	xManualAuto:=ManualAuto, 
	xManualExtend:= 展缸2排液电池阀3手动, 
	xAutoExtend:= 展缸2排液电池阀3自动, 
	xReset:=复位  , 
	xPosExtend:=   , 
	xPosRetract:= , 
	tTimeout:= , 
	yValve1=> 展缸2排液电池阀3, 
	bAlarm=> );	
//展缸2排液电池阀4
cylinder_36(
    xManualRetract := , 
    xAutoRetract := , 
    yValve2 => , 
    cylinder_type :=0 , 

	xManualAuto:=ManualAuto, 
	xManualExtend:= 展缸2排液电池阀4手动, 
	xAutoExtend:= 展缸2排液电池阀4自动, 
	xReset:=复位  , 
	xPosExtend:=   , 
	xPosRetract:= , 
	tTimeout:= , 
	yValve1=> 展缸2排液电池阀4, 
	bAlarm=> );	
//展缸2吹气电池阀1
cylinder_37(
    xManualRetract := , 
    xAutoRetract := , 
    yValve2 => , 
    cylinder_type := 0, 

	xManualAuto:=ManualAuto, 
	xManualExtend:= 展缸2吹气电池阀1手动, 
	xAutoExtend:= 展缸2吹气电池阀1自动, 
	xReset:=复位  , 
	xPosExtend:=   , 
	xPosRetract:= , 
	tTimeout:= , 
	yValve1=> 展缸2吹气电池阀1, 
	bAlarm=> );	
//展缸2吹气电池阀2
cylinder_38(
    xManualRetract := , 
    xAutoRetract := , 
    yValve2 => , 
    cylinder_type := 0, 

	xManualAuto:=ManualAuto, 
	xManualExtend:= 展缸2吹气电池阀2手动, 
	xAutoExtend:= 展缸2吹气电池阀2自动, 
	xReset:=复位  , 
	xPosExtend:=   , 
	xPosRetract:= , 
	tTimeout:= , 
	yValve1=> 展缸2吹气电池阀2, 
	bAlarm=> );	
//展缸1吹气电池阀3
cylinder_39(
    xManualRetract := , 
    xAutoRetract := , 
    yValve2 => , 
    cylinder_type := 0, 

	xManualAuto:=ManualAuto, 
	xManualExtend:= 展缸2吹气电池阀3手动, 
	xAutoExtend:= 展缸2吹气电池阀3自动, 
	xReset:=复位  , 
	xPosExtend:=   , 
	xPosRetract:= , 
	tTimeout:= , 
	yValve1=> 展缸2吹气电池阀3, 
	bAlarm=> );	
//展缸2吹气电池阀4
cylinder_40(
    xManualRetract := , 
    xAutoRetract := , 
    yValve2 => , 
    cylinder_type := 0, 

	xManualAuto:=ManualAuto, 
	xManualExtend:= 展缸2吹气电池阀4手动, 
	xAutoExtend:= 展缸2吹气电池阀4自动, 
	xReset:=复位  , 
	xPosExtend:=   , 
	xPosRetract:= , 
	tTimeout:= , 
	yValve1=> 展缸2吹气电池阀4, 
	bAlarm=> );	
//收集进液电池阀
cylinder_41(
    xManualRetract := , 
    xAutoRetract := , 
    yValve2 => , 
    cylinder_type := 0, 

	xManualAuto:=ManualAuto, 
	xManualExtend:= 收集进液手动, 
	xAutoExtend:= 收集进液自动, 
	xReset:=复位  , 
	xPosExtend:=   , 
	xPosRetract:= , 
	tTimeout:= , 
	yValve1=> 收集平台进液2通电池阀, 
	bAlarm=> );	
//收集排液电池阀
cylinder_42(
    xManualRetract := , 
    xAutoRetract := , 
    yValve2 => , 
    cylinder_type := 0, 

	xManualAuto:=ManualAuto  , 
	xManualExtend:= 收集排液手动, 
	xAutoExtend:= 收集排液自动, 
	xReset:=复位  , 
	xPosExtend:=   , 
	xPosRetract:= , 
	tTimeout:= , 
	yValve1=> 收集平台排液3通电池阀, 
	bAlarm=> );	
//收集正压排液电池阀
cylinder_43(
    xManualRetract := , 
    xAutoRetract := , 
    yValve2 => , 
    cylinder_type :=0 , 

	xManualAuto:=ManualAuto  , 
	xManualExtend:= 收集正压排液手动, 
	xAutoExtend:= 收集正压排液自动, 
	xReset:=复位  , 
	xPosExtend:=   , 
	xPosRetract:= , 
	tTimeout:= , 
	yValve1=> 收集平台正压排液阀, 
	bAlarm=> );	
//溶液收集瓶定位气缸
cylinder_44(
    xManualRetract := , 
    xAutoRetract := , 
    yValve2 => , 
    cylinder_type := 0, 

	xManualAuto:=ManualAuto  , 
	xManualExtend:= 溶液收集瓶定位手动, 
	xAutoExtend:= 溶液收集瓶定位自动, 
	xReset:=复位  , 
	xPosExtend:=   , 
	xPosRetract:= , 
	tTimeout:= , 
	yValve1=> 溶液收集瓶工位定位气缸, 
	bAlarm=> );	
//上样定位气缸
cylinder_45(
    xManualRetract := , 
    xAutoRetract := , 
    yValve2 => , 
    cylinder_type :=0 , 

	xManualAuto:=ManualAuto  , 
	xManualExtend:= 上样定位手动, 
	xAutoExtend:= 上样定位自动, 
	xReset:=复位  , 
	xPosExtend:=   , 
	xPosRetract:= , 
	tTimeout:= , 
	yValve1=> 上样定位气缸, 
	bAlarm=> );	
//上样点样三通电池阀
cylinder_46(
    xManualRetract := , 
    xAutoRetract := , 
    yValve2 => , 
    cylinder_type :=0 , 

	xManualAuto:=ManualAuto  , 
	xManualExtend:= 上样点样三通电池阀手动, 
	xAutoExtend:= 上样点样三通电池阀自动, 
	xReset:=复位  , 
	xPosExtend:=   , 
	xPosRetract:= , 
	tTimeout:= , 
	yValve1=> 上样点样三通电池阀, 
	bAlarm=> );	
//刮板拍照真空泵
cylinder_46(
    xManualRetract := , 
    xAutoRetract := , 
    yValve2 => , 
    cylinder_type := 0, 

	xManualAuto:=ManualAuto  , 
	xManualExtend:=刮板拍照真空手动 , 
	xAutoExtend:= 刮板拍照真空自动, 
	xReset:=复位  , 
	xPosExtend:=   , 
	xPosRetract:= , 
	tTimeout:= , 
	yValve1=> 刮板拍照真空阀, 
	bAlarm=> );	
//刮板拍照无刷电机
cylinder_47(
    xManualRetract := , 
    xAutoRetract := , 
    yValve2 => , 
    cylinder_type :=0 , 

	xManualAuto:=ManualAuto  , 
	xManualExtend:=刮板拍照无刷电机手动 , 
	xAutoExtend:=刮板拍照无刷电机自动 , 
	xReset:=复位  , 
	xPosExtend:=   , 
	xPosRetract:= , 
	tTimeout:= , 
	yValve1=> 刮板拍照无刷电机, 
	bAlarm=> );	
//刮板拍照定位气缸
cylinder_48(
    xManualRetract := , 
    xAutoRetract := , 
    yValve2 => , 
    cylinder_type :=0 , 

	xManualAuto:=ManualAuto  , 
	xManualExtend:= 刮板拍照定位气缸手动, 
	xAutoExtend:=刮板拍照定位气缸自动 , 
	xReset:=复位  , 
	xPosExtend:=   , 
	xPosRetract:= , 
	tTimeout:= , 
	yValve1=> 刮板拍照定位气缸, 
	bAlarm=> );	
//粉末收集器定位气缸
cylinder_49(
    xManualRetract := , 
    xAutoRetract := , 
    yValve2 => , 
    cylinder_type :=0 , 

	xManualAuto:=ManualAuto  , 
	xManualExtend:= 粉末收集器定位手动, 
	xAutoExtend:= 粉末收集器定位自动, 
	xReset:=复位  , 
	xPosExtend:=   , 
	xPosRetract:= , 
	tTimeout:= , 
	yValve1=> 粉末收集器工位定位气缸, 
	bAlarm=> );	
//上样吹气电池阀
cylinder_50(
    xManualRetract := , 
    xAutoRetract := , 
    yValve2 => , 
    cylinder_type := 0, 

	xManualAuto:=ManualAuto  , 
	xManualExtend:= 上样吹气手动, 
	xAutoExtend:= 上样吹气自动, 
	xReset:=复位  , 
	xPosExtend:=   , 
	xPosRetract:= , 
	tTimeout:= , 
	yValve1=> 上样吹气二通阀, 
	bAlarm=> );

END_PROGRAM

// Device/Application/25_FB_功能块/FB_cylinder
FUNCTION_BLOCK FB_cylinder
VAR_INPUT
    xManualAuto : BOOL := FALSE;  // 手自动模式：FALSE=手动，TRUE=自动
    xManualExtend : BOOL;  // 手动伸出
	// 手动缩回
	xManualRetract: BOOL;
    xAutoExtend : BOOL;  // 自动伸出
	// 自动缩回
	xAutoRetract: BOOL;
    xReset : BOOL;  // 复位按钮
    xPosExtend : BOOL;  // 伸出到位传感器
    xPosRetract : BOOL;  // 缩回到位传感器
    tTimeout : TIME := T#5S;  // 动作超时时间
END_VAR
VAR_OUTPUT
    yValve1 : BOOL;  // 电磁阀1输出：TRUE=伸出，FALSE=缩回
	// 电磁阀2输出：TRUE=伸出，FALSE=缩回
	yValve2: BOOL;
    bAlarm : BOOL;  // 报警输出
END_VAR
VAR
    bEnableCmd1 : BOOL;  // 有效的命令1
	// 有效的命令1
	bEnableCmd2: BOOL;
	tActionTimer: TON;// 动作定时器
END_VAR
VAR_INPUT
	// 气缸类型  0 单控  1双控
	cylinder_type: INT;
END_VAR



CASE cylinder_type OF
	0:     //单控电池阀
		//命令逻辑选择
		IF xManualAuto  THEN
			//自动模式，使用自动命令
			bEnableCmd1 :=xAutoExtend;
			ELSE
			//手动模式，使用手动命令
			bEnableCmd1 :=xManualExtend  ;
		END_IF
		//控制指令
		IF bEnableCmd1 THEN
			//开始伸出
			yValve1:=TRUE;
			ELSE
			//开始缩回
			yValve1 :=FALSE;
		END_IF
		
	
			tActionTimer(IN := (NOT xPosExtend AND NOT yValve1)  OR   (NOT xPosRetract AND yValve1), PT:=tTimeout );
			bAlarm :=tActionTimer .Q;
	
	1:        //双控电池阀
		//命令逻辑选择
		IF xManualAuto  THEN
			//自动模式，使用自动命令
			bEnableCmd1 :=xAutoExtend;
			bEnableCmd2 :=xAutoRetract;
		ELSE
			//手动模式，使用手动命令
			bEnableCmd1 :=xManualExtend;
			bEnableCmd2 :=xManualRetract;
		END_IF
		//伸出控制指令
		IF bEnableCmd1 THEN
			//开始伸出
			yValve1:=TRUE;
			yValve2:=FALSE;
		ELSE 
			yValve1:=FALSE;
		END_IF
		
		IF bEnableCmd2 THEN
			//开始缩回
			yValve2:=TRUE;
			yValve1:=FALSE;
		ELSE 
			yValve2:=FALSE;
		END_IF
		
			tActionTimer(IN := (NOT xPosExtend AND NOT yValve1)  OR   (NOT xPosRetract AND yValve2), PT:=tTimeout );
			bAlarm :=tActionTimer .Q;
		
END_CASE

IF xReset THEN
	bAlarm:=FALSE ;
END_IF

END_FUNCTION_BLOCK

// Device/Application/50_action/Rail_Sync
PROGRAM Rail_Sync
VAR
	i : INT;
END_VAR

(* 地轨 11Y 双源同步桥 (非动作派发器, 是 PC<->HMI 点位对账工具).
   原理: HMI_地轨轴11Y.position[] 是单 ExtensionObject struct, OPC 逐成员读写不可行
         -> 让 PLC 当桥, OPC 只暴露 flat 数组 (复用 *_ActPos 镜像同套路).
   每扫描无条件执行 (挂 PLC_MainPRG 无条件段, 与 ActPos 镜像同处; 勿放运行态 CASE).
   守恒: PUSH 纯 PLC 内存拷贝, 任一侧可触发; PULL 写真源恒为 PC, HMI 触发=请 PC 提交. *)

// (1) 常开镜像: HMI 教值 -> flat 只读镜像 (PC 经此读做 diff/pull, 不直访 struct)
FOR i := 1 TO 6 DO
	Rail_Pos_HMI[i] := HMI_地轨轴11Y.position[i];
END_FOR

// (2) 同步邮箱
CASE Rail_Sync_Req OF
	1:  (* PUSH: PC 真源 Rail_Pos_Target[] -> HMI 工作副本 position[] (PLC 写自己 struct, 无 OPC 限制) *)
		FOR i := 1 TO 6 DO
			HMI_地轨轴11Y.position[i] := Rail_Pos_Target[i];
		END_FOR
		Rail_Sync_Ack := 1;     (* 完成 *)
		Rail_Sync_Req := 0;     (* 清请求 *)

	2:  (* PULL: 收现场教值回真源. PLC 写不了 yaml, 更不可碰 Rail_Pos_Target (单写者=PC).
	          -> 仅亮邮箱待 PC 提交. PC 轮询见 Req=2 -> 读 Rail_Pos_HMI[] -> 限位校验/diff/确认
	             -> 写 points.yaml + 重算并写 Rail_Pos_Target[] -> 由 PC 置 Req:=0,Ack:=1 (失败 Ack:=3). *)
		Rail_Sync_Ack := 2;     (* 待 PC 提交 (PC 接手后由 PC 改写 Ack/Req) *)
END_CASE

END_PROGRAM

// Device/Application/50_action/PLC_Pump_泵管理
PROGRAM PLC_Pump_泵管理
VAR
END_VAR

(* 真空泵集中管理: 大真空泵线圈的唯一聚合点 (每扫描无条件调用).
   大真空泵站位[] 引用计数总线 -> 大真空泵自动 (经 FB_cylinder cylinder_8 驱动 大真空泵 %QX2.4).
   写者: [0..8]=Develop_TankDrain 排液自治; [11]=上位机 Pump_L2 显式真空; [9][10] 已退役. *)
大真空泵自动 := 大真空泵站位[0] OR 大真空泵站位[1] OR 大真空泵站位[2] OR 大真空泵站位[3]
	OR 大真空泵站位[4] OR 大真空泵站位[5] OR 大真空泵站位[6] OR 大真空泵站位[7]
	OR 大真空泵站位[8] OR 大真空泵站位[9] OR 大真空泵站位[10] OR 大真空泵站位[11];

END_PROGRAM

// Device/Application/40_Man/Develop_TankDrain
PROGRAM Develop_TankDrain
VAR
	// 循环索引
	i: INT;
	// 全局真空泵控制标志
	anyDraining: BOOL;
	// 全局真空泵控制标志
	展开step: INT;
	// 全局真空泵控制标志
	TON_3: TON;
	// 全局真空泵控制标志
	TON_4: TON;
	BlowTimer: ARRAY[1..8] OF TON;
	BlowDuration: TIME := TIME#30s0ms;
END_VAR




A50_Expand_liquid_discharge_排液();

ACTION A50_Expand_liquid_discharge_排液:

// ══════════════════════════════════════════════════════════════
// 排液控制程序（per-tank 并行 FSM，每扫描周期调用）
// ══════════════════════════════════════════════════════════════
// 程序名：PRG_TankDrain
// 文件名：plc_develop_drain.txt
// 职责：监控 Tank_Drain_Enable[1..8]，触发对应缸的 3 阶段排液流程
// 触发条件：Tank_Drain_Enable[i]=TRUE 且 Tank_State[i]=40
// 完成标志：Tank_Drain_Done[i]=TRUE, Tank_State[i]=99
// 复位方式：PC 写 Tank_Drain_Enable[i]=FALSE → 清 Done；
//           PC 写 Tank_State[i]=0 → 释放缸
// ══════════════════════════════════════════════════════════════
// 3 阶段排液时序（工程师已验证）：
//   Phase A — Draining(50)：开排液阀 + 真空泵，等待 DrainDuration
//   Phase B — BlowAir(55) ：追加开吹气阀，等待 BlowDuration
//   Phase C — CylinderRetract(60)：关所有阀 + 气缸退回，等待到位传感器
// ══════════════════════════════════════════════════════════════
// 硬件拓扑：
//   - 每缸有独立排液电磁阀、吹气电磁阀、气缸（伸出/退回）
//   - 真空泵（大真空泵）全局共享，anyDraining 引用计数式控制
//   - 排液气泡传感器按组共享（仅用于监控，不参与控制逻辑）
//   - 支持 8 缸完全并行排液（各缸 FSM 独立推进）
// ══════════════════════════════════════════════════════════════
// Tank_State 状态转换（排液相关）：
//   40 (Developing)      → 50 (Draining)        : Drain_Enable[i] 触发
//   50 (Draining)        → 55 (BlowAir)         : DrainTimer[i].Q
//   55 (BlowAir)         → 60 (CylinderRetract) : BlowTimer[i].Q
//   60 (CylinderRetract) → 99 (Done)            : 气缸到位传感器
//   99 (Done)            → 0  (Idle)            : PC 写 Tank_State=0
//   50/55/60             → 90 (Error)           : 急停
//   注：55/60 为 PLC 内部子状态，PC 只关心 Drain_Done（state 99）
// ══════════════════════════════════════════════════════════════
// 物理 IO 映射表（工程师变量名 → 缸索引）：
//   i=1: 展缸1排液电池阀1自动 / 展缸1吹气电池阀1自动 / 展缸1气缸1自动 / 展缸1气缸1动点
//   i=2: 展缸1排液电池阀2自动 / 展缸1吹气电池阀2自动 / 展缸1气缸2自动 / 展缸1气缸2动点
//   i=3: 展缸1排液电池阀3自动 / 展缸1吹气电池阀3自动 / 展缸1气缸3自动 / 展缸1气缸3动点
//   i=4: 展缸1排液电池阀4自动 / 展缸1吹气电池阀4自动 / 展缸1气缸4自动 / 展缸1气缸4动点
//   i=5: 展缸2排液电池阀1自动 / 展缸2吹气电池阀1自动 / 展缸2气缸1自动 / 展缸2气缸1动点
//   i=6: 展缸2排液电池阀2自动 / 展缸2吹气电池阀2自动 / 展缸2气缸2自动 / 展缸2气缸2动点
//   i=7: 展缸2排液电池阀3自动 / 展缸2吹气电池阀3自动 / 展缸2气缸3自动 / 展缸2气缸3动点
//   i=8: 展缸2排液电池阀4自动 / 展缸2吹气电池阀4自动 / 展缸2气缸4自动 / 展缸2气缸4动点
//   全局: 大真空泵自动
//   监控: 展缸1排液气泡传感器 / 展缸2排液气泡传感器
// ══════════════════════════════════════════════════════════════



// ══ 急停联锁：排液程序响应急停 ══
IF NOT 急停 THEN
    FOR i := 1 TO 8 DO
        // 急停时将所有排液中的缸（50/55/60）标记为 Error
        IF Tank_State[i] = 50 OR Tank_State[i] = 55 OR Tank_State[i] = 60 THEN
            Tank_State[i] := 90;
        END_IF
        // 停止所有定时器
        DrainTimer[i](IN := FALSE, PT := T#0S);
        BlowTimer[i](IN := FALSE, PT := T#0S);
        // 关闭所有排液阀和吹气阀
        CASE i OF
            1: 展缸1排液电池阀1自动 := FALSE; 展缸1吹气电池阀1自动 := FALSE;
            2: 展缸1排液电池阀2自动 := FALSE; 展缸1吹气电池阀2自动 := FALSE;
            3: 展缸1排液电池阀3自动 := FALSE; 展缸1吹气电池阀3自动 := FALSE;
            4: 展缸1排液电池阀4自动 := FALSE; 展缸1吹气电池阀4自动 := FALSE;
            5: 展缸2排液电池阀1自动 := FALSE; 展缸2吹气电池阀1自动 := FALSE;
            6: 展缸2排液电池阀2自动 := FALSE; 展缸2吹气电池阀2自动 := FALSE;
            7: 展缸2排液电池阀3自动 := FALSE; 展缸2吹气电池阀3自动 := FALSE;
            8: 展缸2排液电池阀4自动 := FALSE; 展缸2吹气电池阀4自动 := FALSE;
        END_CASE
    END_FOR
    // 关闭真空泵
    大真空泵站位[0] := FALSE;
    RETURN;
END_IF

// ══ 主循环：逐缸并行处理排液 FSM ══
FOR i := 1 TO 8 DO
 DrainTimer[i](IN := (Tank_State[i] = 50  AND  (i>4 AND 展缸2溶剂废液检测传感器)) OR (Tank_State[i] = 50 AND (i<5 AND 展缸1溶剂废液检测传感器)) , PT := DrainDuration);

 BlowTimer[i](IN := Tank_State[i] = 55, PT := BlowDuration);
 
    // ── 场景 1：PC 撤销 Drain_Enable → 复位 Done 标志（握手完成）──
    IF NOT Tank_Drain_Enable[i] THEN
        Tank_Drain_Done[i] := FALSE;
        DrainTimer[i](IN := FALSE, PT := T#0S);
        BlowTimer[i](IN := FALSE, PT := T#0S);
        // 注意：不主动修改 Tank_State，由 PC 写 0 释放
    // ── 场景 2：Drain_Enable=TRUE，缸处于 Developing(40)，启动排液 Phase A ──
    ELSIF Tank_Drain_Enable[i] AND Tank_State[i] = 40 THEN
        // 开启排液阀
		大真空泵站位[i] := TRUE;
        CASE i OF
            1: 展缸1排液电池阀1自动 := TRUE;
            2: 展缸1排液电池阀2自动 := TRUE;
            3: 展缸1排液电池阀3自动 := TRUE;
            4: 展缸1排液电池阀4自动 := TRUE;
            5: 展缸2排液电池阀1自动 := TRUE;
            6: 展缸2排液电池阀2自动 := TRUE;
            7: 展缸2排液电池阀3自动 := TRUE;
            8: 展缸2排液电池阀4自动 := TRUE;
        END_CASE
        // 推进状态至 Draining
        Tank_State[i] := 50;
    // ── 场景 3：Phase A — Draining(50)，排液阀开 + 真空泵运行，等待排液定时完成 ──
    ELSIF Tank_State[i] = 50 AND (i<5 AND 展缸1溶剂废液检测传感器) THEN
       
        IF DrainTimer[i].Q THEN
            // 排液定时完成，锁定并复位 DrainTimer
            DrainTimer[i](IN := FALSE, PT := T#0S);
            // 开启吹气阀（排液阀保持开启），进入 Phase B
            CASE i OF
                1: 展缸1吹气电池阀1自动 := TRUE;
                2: 展缸1吹气电池阀2自动 := TRUE;
                3: 展缸1吹气电池阀3自动 := TRUE;
                4: 展缸1吹气电池阀4自动 := TRUE;
                
            END_CASE
            Tank_State[i] := 55;
        END_IF
	ELSIF Tank_State[i] = 50  AND  (i>4AND 展缸2溶剂废液检测传感器) THEN
       
        IF DrainTimer[i].Q THEN
            // 排液定时完成，锁定并复位 DrainTimer
            DrainTimer[i](IN := FALSE, PT := T#0S);
            // 开启吹气阀（排液阀保持开启），进入 Phase B
            CASE i OF
                5: 展缸2吹气电池阀1自动 := TRUE;
                6: 展缸2吹气电池阀2自动 := TRUE;
                7: 展缸2吹气电池阀3自动 := TRUE;
                8: 展缸2吹气电池阀4自动 := TRUE;
            END_CASE
            Tank_State[i] := 55;
        END_IF
    // ── 场景 4：Phase B — BlowAir(55)，吹气阀开，等待吹气定时完成 ──
    ELSIF Tank_State[i] = 55 THEN
        大真空泵站位[i] := FALSE;
        IF BlowTimer[i].Q THEN
            // 吹气完成，锁定并复位 BlowTimer
            BlowTimer[i](IN := FALSE, PT := T#0S);
            // 关闭排液阀和吹气阀，启动气缸退回，进入 Phase C
            CASE i OF
                1: 展缸1排液电池阀1自动 := FALSE; 展缸1吹气电池阀1自动 := FALSE; 展缸1气缸1自动 := FALSE;
                2: 展缸1排液电池阀2自动 := FALSE; 展缸1吹气电池阀2自动 := FALSE; 展缸1气缸2自动 := FALSE;
                3: 展缸1排液电池阀3自动 := FALSE; 展缸1吹气电池阀3自动 := FALSE; 展缸1气缸3自动 := FALSE;
                4: 展缸1排液电池阀4自动 := FALSE; 展缸1吹气电池阀4自动 := FALSE; 展缸1气缸4自动 := FALSE;
                5: 展缸2排液电池阀1自动 := FALSE; 展缸2吹气电池阀1自动 := FALSE; 展缸2气缸1自动 := FALSE;
                6: 展缸2排液电池阀2自动 := FALSE; 展缸2吹气电池阀2自动 := FALSE; 展缸2气缸2自动 := FALSE;
                7: 展缸2排液电池阀3自动 := FALSE; 展缸2吹气电池阀3自动 := FALSE; 展缸2气缸3自动 := FALSE;
                8: 展缸2排液电池阀4自动 := FALSE; 展缸2吹气电池阀4自动 := FALSE; 展缸2气缸4自动 := FALSE;
            END_CASE
            Tank_State[i] := 60;
       END_IF
    // ── 场景 5：Phase C — CylinderRetract(60)，等待气缸退回到位 ──
    ELSIF Tank_State[i] = 60 THEN
        CASE i OF
            1: IF 展缸1气缸1原点 THEN   Tank_Drain_Done[1] := TRUE; Tank_State[1] := 99; END_IF
            2: IF 展缸1气缸2原点 THEN   Tank_Drain_Done[2] := TRUE; Tank_State[2] := 99; END_IF
            3: IF 展缸1气缸3原点 THEN   Tank_Drain_Done[3] := TRUE; Tank_State[3] := 99; END_IF
            4: IF 展缸1气缸4原点 THEN   Tank_Drain_Done[4] := TRUE; Tank_State[4] := 99; END_IF
            5: IF 展缸2气缸1原点 THEN   Tank_Drain_Done[5] := TRUE; Tank_State[5] := 99; END_IF
            6: IF 展缸2气缸2原点 THEN   Tank_Drain_Done[6] := TRUE; Tank_State[6] := 99; END_IF
            7: IF 展缸2气缸3原点 THEN   Tank_Drain_Done[7] := TRUE; Tank_State[7] := 99; END_IF
            8: IF 展缸2气缸4原点 THEN   Tank_Drain_Done[8] := TRUE; Tank_State[8] := 99; END_IF
        END_CASE
	END_IF
END_FOR
END_ACTION

END_PROGRAM

// Device/Application/50_action/Pump_L2
PROGRAM Pump_L2
VAR
	bActionDone: BOOL;
	bActionError: BOOL;
	L2_StartTrig: R_TRIG;
END_VAR

(* Pump 真空泵 L2 统一动作派发器 (独立真空泵原子动作通道).
   按 Pump_L2_ActionCode 派发: 10=真空泵开 / 20=真空泵关; 写上位机泵槽 大真空泵站位[11].
   实际线圈由 PLC_Pump_泵管理 聚合 大真空泵站位[] 驱动.
   Start 上升沿接受 -> RUNNING 调原子 -> bActionDone=DONE. *)
L2_StartTrig(CLK := Pump_L2_Start);

CASE Pump_L2_State OF
	0:  (* IDLE *)
		Pump_L2_Step := 0;
		IF L2_StartTrig.Q THEN
			Pump_L2_AcceptedSeq := Pump_L2_RequestSeq;
			Pump_L2_ActiveCode  := Pump_L2_ActionCode;
			Pump_L2_ErrorCode   := 0;
			Pump_L2_Retryable   := FALSE;
			bActionDone  := FALSE;
			bActionError := FALSE;
			CASE Pump_L2_ActionCode OF
				10, 20:
					Pump_L2_SafeState := 0;
					Pump_L2_State     := 10;   (* RUNNING *)
			ELSE
				Pump_L2_ErrorCode    := 101;  (* 未知动作码 *)
				Pump_L2_Retryable    := TRUE;
				Pump_L2_CompletedSeq := Pump_L2_AcceptedSeq;
				Pump_L2_State        := 30;   (* REJECTED *)
			END_CASE
		END_IF

	10: (* RUNNING *)
		IF Pump_L2_Reset THEN                (* RUNNING 中 RESET: 中止回 IDLE *)
			Pump_L2_State := 0;
		ELSE
			CASE Pump_L2_ActiveCode OF
				10: A10_vacuum_on();
				20: A20_vacuum_off();
			END_CASE
			IF bActionDone THEN
				bActionDone          := FALSE;
				Pump_L2_CompletedSeq := Pump_L2_AcceptedSeq;
				Pump_L2_State        := 20;   (* DONE *)
			ELSIF bActionError THEN
				bActionError         := FALSE;
				Pump_L2_Retryable    := TRUE;
				Pump_L2_CompletedSeq := Pump_L2_AcceptedSeq;
				Pump_L2_State        := 40;   (* ERROR *)
			END_IF
		END_IF

	20, 30, 40, 50:  (* 终态: 等 Start 落沿或 Reset 回 IDLE *)
		IF (NOT Pump_L2_Start) OR Pump_L2_Reset THEN
			Pump_L2_State := 0;
		END_IF
END_CASE

ACTION A10_vacuum_on:
(* 真空泵开: 置上位机泵槽 (实际线圈由 PLC_Pump_泵管理 聚合 大真空泵站位[] 驱动) *)
大真空泵站位[11] := TRUE;
bActionDone := TRUE;
END_ACTION

ACTION A20_vacuum_off:
(* 真空泵关: 清上位机泵槽 (排液 [0..8] 仍可独立保持真空) *)
大真空泵站位[11] := FALSE;
bActionDone := TRUE;
END_ACTION

END_PROGRAM

// Device/Application/50_action/Rail_L2
PROGRAM Rail_L2
VAR
	L2_StartTrig : R_TRIG;
	fTgt: LREAL;
END_VAR

(* 地轨 11Y L2 统一动作派发器 (第7通道).
   按位置码移地轨: Rail_L2_ActionCode=10 -> 移到 Rail_Pos_Target[Rail_Target_Position] (1..6, PC 真源).
   地轨坐标真源已收编为 PC 写的 Rail_Pos_Target[]; HMI position[] 降为手动示教工作副本, 自动不再读它.
   Start 上升沿接受 -> RUNNING 下发移动 -> bAbMoveDone=DONE. *)
L2_StartTrig(CLK := Rail_L2_Start);

CASE Rail_L2_State OF
	0:  (* IDLE *)
		Rail_L2_Step := 0;
		IF L2_StartTrig.Q THEN
			Rail_L2_AcceptedSeq := Rail_L2_RequestSeq;
			Rail_L2_ActiveCode  := Rail_L2_ActionCode;
			Rail_L2_ErrorCode   := 0;
			Rail_L2_Retryable   := FALSE;
// 			IF Rail_L2_ActionCode = 10
// 			   AND Rail_Target_Position >= 1 AND Rail_Target_Position <= 6 THEN
// 				Rail_L2_SafeState := 0;
// // 				地轨轴11YDATE.fAbsTarget := HMI_地轨轴11Y.position[Rail_Target_Position];
// 				地轨轴11YDATE.fAbsTarget := Rail_Pos_Target[Rail_Target_Position];
// 				地轨轴11YDATE.xMoveAbs   := TRUE;
// 				Rail_L2_State := 10;   (* RUNNING *)
// 			ELSE
// 				Rail_L2_ErrorCode    := 101;  (* 未知动作码 / 非法位置码 *)
// 				Rail_L2_Retryable    := TRUE;
// 				Rail_L2_CompletedSeq := Rail_L2_AcceptedSeq;
// 				Rail_L2_State        := 30;   (* REJECTED *)
// 			END_IF
			IF Rail_L2_ActionCode = 10 AND Rail_Target_Position >= 1 AND Rail_Target_Position <= 6 THEN
				fTgt := Rail_Pos_Target[Rail_Target_Position];     (* PC 真源坐标 *)
				IF fTgt <= 0.0 OR fTgt > 3000.0 THEN
					(* 兜底: PC 未 push / 重启后 Rail_Pos_Target 归 0 / 越限 → 拒绝, 绝不移到 0 端 *)
					Rail_L2_ErrorCode    := 102;   (* 目标未初始化或越限 *)
					Rail_L2_Retryable    := TRUE;
					Rail_L2_CompletedSeq := Rail_L2_AcceptedSeq;
					Rail_L2_State        := 30;    (* REJECTED *)
				ELSE
					Rail_L2_SafeState        := 0;
					地轨轴11YDATE.fAbsTarget := fTgt;
					地轨轴11YDATE.xMoveAbs   := TRUE;
					Rail_L2_State            := 10; (* RUNNING *)
				END_IF
			ELSE
				Rail_L2_ErrorCode    := 101;   (* 未知动作码 / 非法位置码 *)
				Rail_L2_Retryable    := TRUE;
				Rail_L2_CompletedSeq := Rail_L2_AcceptedSeq;
				Rail_L2_State        := 30;    (* REJECTED *)
END_IF
		END_IF

	10: (* RUNNING *)
		IF Rail_L2_Reset THEN                 (* RUNNING 中 RESET: 中止回 IDLE *)
			地轨轴11YDATE.xMoveAbs := FALSE;
			Rail_L2_State := 0;
		ELSIF 地轨轴11YDATE.bAbMoveDone THEN
			地轨轴11YDATE.xMoveAbs   := FALSE;
			Rail_L2_CompletedSeq := Rail_L2_AcceptedSeq;
			Rail_L2_State        := 20;   (* DONE *)
		END_IF
		(* 如地轨伺服有报警位, 在此 ELSIF <报警> THEN 置 Rail_L2_ErrorCode + State:=40 *)

	20, 30, 40, 50:  (* 终态: 等 Start 落沿或 Reset 回 IDLE *)
		IF (NOT Rail_L2_Start) OR Rail_L2_Reset THEN
			Rail_L2_State := 0;
		END_IF
END_CASE

END_PROGRAM

// Device/Application/50_action/FeedLift_L2
PROGRAM FeedLift_L2
VAR
	上料step: INT;
	下料step: INT;
	bActionDone: BOOL;
	bActionError: BOOL;
	L2_StartTrig: R_TRIG;
	feedlift_TO: TON;
END_VAR

(* FeedLift 工位 L2 统一动作派发器
   按 FeedLift_L2_ActionCode 派发到纯设备原子动作 (不含机器人/相机/CNC 握手).
   Start 上升沿接受请求 -> RUNNING 每周期调用对应原子 -> bActionDone=DONE / bActionError=ERROR. *)
L2_StartTrig(CLK := FeedLift_L2_Start);

CASE FeedLift_L2_State OF
	0:  (* IDLE *)
		FeedLift_L2_Step := 0;
		IF L2_StartTrig.Q THEN
			FeedLift_L2_AcceptedSeq := FeedLift_L2_RequestSeq;
			FeedLift_L2_ActiveCode  := FeedLift_L2_ActionCode;
			FeedLift_L2_ErrorCode   := 0;
			FeedLift_L2_Retryable   := FALSE;
			bActionDone  := FALSE;
			bActionError := FALSE;
			上料step := 0;
			下料step := 0;
			CASE FeedLift_L2_ActionCode OF
				11, 12, 21, 22:
					FeedLift_L2_SafeState := 0;
					FeedLift_L2_State     := 10;   (* RUNNING *)
			ELSE
				FeedLift_L2_ErrorCode    := 101;  (* 未知动作码 *)
				FeedLift_L2_Retryable    := TRUE;
				FeedLift_L2_CompletedSeq := FeedLift_L2_AcceptedSeq;
				FeedLift_L2_State        := 30;   (* REJECTED *)
			END_CASE
		END_IF

	10: (* RUNNING *)
		IF FeedLift_L2_Reset THEN FeedLift_L2_State := 0; RETURN; END_IF   (* RUNNING 中 RESET: 中止挂死动作 *)
		CASE FeedLift_L2_ActiveCode OF
			11: A11_feed_raise();
			12: A12_feed_lower();
			21: A21_unload_ready();
			22: A22_unload_bury();
		END_CASE
		IF bActionDone THEN
			bActionDone              := FALSE;
			FeedLift_L2_CompletedSeq := FeedLift_L2_AcceptedSeq;
			FeedLift_L2_State        := 20;   (* DONE *)
		ELSIF bActionError THEN              (* 设备预条件未满足 -> 报错交上位机 *)
			bActionError             := FALSE;
			FeedLift_L2_Retryable    := TRUE;
			FeedLift_L2_CompletedSeq := FeedLift_L2_AcceptedSeq;
			FeedLift_L2_State        := 40;   (* ERROR; ErrorCode 由原子置 *)
		END_IF

	20, 30, 40, 50:  (* 终态: 等 Start 落沿或 Reset 回 IDLE *)
		IF (NOT FeedLift_L2_Start) OR FeedLift_L2_Reset THEN
			FeedLift_L2_State := 0;
		END_IF
END_CASE

ACTION A11_feed_raise:
(* 上料: jog 上料Z1 升至取料光电 (上位机随后驱动机器人吸料); 无玻璃则报错交上位机 *)
feedlift_TO(IN:=上料step=0, PT:=T#10S);
CASE 上料step OF
	0:
		IF 玻璃上料轴1ZDATE.bHomed AND 玻璃升降接近开关1 AND 上料进料传感器 AND NOT Alarm.0 THEN
			上料step:=1;
		ELSIF feedlift_TO.Q THEN
			FeedLift_L2_ErrorCode:=301;   (* 上料无玻璃/传感器未就绪 *)
			上料step:=0;
			bActionError:=TRUE;
		END_IF
	1:
		IF 玻璃上料轴1ZDATE.fActPos>=510.0 AND 玻璃升降光电开关1 AND NOT 玻璃升降接近开关1 THEN
			Z1JOG_pos:=FALSE;
			Alarm.0:=TRUE;                       (* 上料机构无玻璃 *)
			上料step:=0;
			FeedLift_L2_ErrorCode:=301;
			bActionError:=TRUE;
		ELSIF NOT 玻璃升降光电开关1 AND 玻璃上料轴1ZDATE.fActPos<514 THEN
			Z1JOG_pos:=TRUE;
		ELSE
			Z1JOG_pos:=FALSE;
			上料step:=0;
			bActionDone:=TRUE;
		END_IF
END_CASE
END_ACTION

ACTION A22_unload_bury:
(* 下料: 机器人放废料后, jog Z2 下埋至光电消失 *)
feedlift_TO(IN:=下料step=0, PT:=T#10S);
CASE 下料step OF
	0:
		IF 玻璃升降光电开关2 AND 玻璃升降接近开关2 THEN
			Z2JOG_NEG:=TRUE;
			下料step:=10;
		ELSIF feedlift_TO.Q THEN
			FeedLift_L2_ErrorCode:=302;   (* 下料无玻璃/传感器未就绪 *)
			下料step:=0;
			bActionError:=TRUE;
		END_IF
	10:
		IF NOT 玻璃升降光电开关2 THEN
			Z2JOG_NEG:=FALSE;
			下料step:=0;
			bActionDone:=TRUE;
		END_IF
END_CASE
END_ACTION

ACTION A12_feed_lower:
(* 上料: 机器人吸住玻璃后, Z1 相对下降 5mm 让位 *)
CASE 上料step OF
	0:
		玻璃上料轴1ZDATE.fRelTarget:=-5.0;
		玻璃上料轴1ZDATE.xMoveRel:=TRUE;
		上料step:=10;
	10:
		IF 玻璃上料轴1ZDATE.bReMoveDone THEN
			玻璃上料轴1ZDATE.xMoveRel:=FALSE;
			上料step:=0;
			bActionDone:=TRUE;
		END_IF
END_CASE
END_ACTION

ACTION A21_unload_ready:
(* 下料: jog 下料Z2 到放废料位 (上位机随后驱动机器人放废料) *)
CASE 下料step OF
	0:
		IF 玻璃上料轴2ZDATE.bHomed AND 下料出料传感器 AND NOT Alarm.1 THEN
			下料step:=1;
		END_IF
	1:
		IF NOT 玻璃升降光电开关2 AND 玻璃上料轴2ZDATE.fActPos<510 THEN
			Z2JOG_POS:=TRUE;
		ELSE
			Z2JOG_POS:=FALSE;
			下料step:=10;
		END_IF
	10:
		IF 玻璃升降光电开关2 THEN
			Z2JOG_NEG:=TRUE;
			下料step:=15;
		END_IF
	15:
		IF NOT 玻璃升降光电开关2 THEN
			Z2JOG_NEG:=FALSE;
			下料step:=0;
			bActionDone:=TRUE;
		END_IF
END_CASE
END_ACTION

END_PROGRAM

// Device/Application/50_action/Sampling_L2
PROGRAM Sampling_L2
VAR
	初始化step: INT;
	清洗step: INT;
	清洗计数: INT;
	放硅胶板STEP: INT;
	上样准备step: INT;
	吸收液体step: INT;
	点样step: INT;
	喷涂移轴step: INT;
	N: INT;
	A: INT;
	打样伺服移动step: INT;
	spot_band_step: INT;
	spot_band_dry_count: INT;
	spot_band_old_6x_velocity: LREAL;
	spot_band_velocity_saved: BOOL;
	bActionDone: BOOL;
	bActionError: BOOL;
	TON_0: TON;
	TON_1: TON;
	L2_StartTrig: R_TRIG;
	R_TRIG: ARRAY[1..12] OF R_TRIG;
	TON: ARRAY[1..11] OF TON;
END_VAR

(* Sampling 工位 L2 统一动作派发器
   按 Sampling_L2_ActionCode 派发到纯设备原子动作 (不含机器人/相机/CNC 握手).
   Start 上升沿接受请求 -> RUNNING 每周期调用对应原子 -> bActionDone=DONE / bActionError=ERROR. *)
L2_StartTrig(CLK := Sampling_L2_Start);

CASE Sampling_L2_State OF
	0:  (* IDLE *)
		Sampling_L2_Step := 0;
		IF L2_StartTrig.Q THEN
			Sampling_L2_AcceptedSeq := Sampling_L2_RequestSeq;
			Sampling_L2_ActiveCode  := Sampling_L2_ActionCode;
			Sampling_L2_ErrorCode   := 0;
			Sampling_L2_Retryable   := FALSE;
			bActionDone  := FALSE;
			bActionError := FALSE;
			初始化step := 0;
			清洗step := 0;
			放硅胶板STEP := 0;
			上样准备step := 0;
			吸收液体step := 0;
			点样step := 0;
			喷涂移轴step := 0;
			spot_band_step := 0;
			spot_band_dry_count := 0;
			spot_band_velocity_saved := FALSE;
			CASE Sampling_L2_ActionCode OF
				10, 20, 31, 32, 33, 40, 50, 60, 61, 62:
					Sampling_L2_SafeState := 0;
					Sampling_L2_State     := 10;   (* RUNNING *)
			ELSE
				Sampling_L2_ErrorCode    := 101;  (* 未知动作码 *)
				Sampling_L2_Retryable    := TRUE;
				Sampling_L2_CompletedSeq := Sampling_L2_AcceptedSeq;
				Sampling_L2_State        := 30;   (* REJECTED *)
			END_CASE
		END_IF

	10: (* RUNNING *)
		IF Sampling_L2_Reset THEN
			IF Sampling_L2_ActiveCode = 62 THEN
				上样点样三通电池阀自动 := FALSE;
				上样吹气自动 := FALSE;
				点样轴6XDATE.xMoveAbs := FALSE;
				点样轴7YDATE.xMoveAbs := FALSE;
				泵站位符 := FALSE;
				IF spot_band_velocity_saved THEN
					点样轴6XDATE.fVelocity := spot_band_old_6x_velocity;
					spot_band_velocity_saved := FALSE;
				END_IF
				spot_band_step := 0;
			END_IF
			Sampling_L2_State := 0;
			RETURN;
		END_IF   (* RUNNING ? RESET: ?????? *)
		CASE Sampling_L2_ActiveCode OF
			10: A10_init_初始化();
			20: A20_clean_清洗();
			31: A31_放板移轴();
			32: A32_放板定位();
			33: (* 定位松开: 松开上样定位气缸释放硅胶板 (上位机随后驱动机器人取板); 镜像 A32 放板定位 *)
				上样定位自动 := FALSE;
				bActionDone := TRUE;
			40: A40_prep_上样准备();
			50: A50_absorb_吸收液体();
			60: A60_spray_点样();
			61: (* 喷涂移轴: 点样7Y轴移入喷涂位 (HMI 示教 position[2]); 镜像 A31 放板移轴 *)
				CASE 喷涂移轴step OF
					0:
						点样轴7YDATE.fAbsTarget := HMI_点样轴7Y.position[2];
						点样轴7YDATE.xMoveAbs := TRUE;
						喷涂移轴step := 10;
					10:
						IF 点样轴7YDATE.bAbMoveDone THEN
							点样轴7YDATE.xMoveAbs := FALSE;
							喷涂移轴step := 0;
							bActionDone := TRUE;
						END_IF
				END_CASE
			62: (* ?????+????: 6X ???? PLC ??? T ??; ??? ON ???/????? *)
				Sampling_L2_Step := spot_band_step;
				CASE spot_band_step OF
					0:
						IF NOT spot_band_velocity_saved THEN
							spot_band_old_6x_velocity := 点样轴6XDATE.fVelocity;
							spot_band_velocity_saved := TRUE;
						END_IF
						IF Sampling_band_dry_cycles < 1 THEN
							Sampling_band_dry_cycles := 1;
						END_IF
						点样轴6XDATE.xMoveAbs := FALSE;
						点样轴7YDATE.xMoveAbs := FALSE;
						上样点样三通电池阀自动 := FALSE;
						上样吹气自动 := FALSE;
						IF Sampling_band_spot_speed > 0.0 THEN
							点样轴6XDATE.fVelocity := Sampling_band_spot_speed;
						END_IF
						点样轴6XDATE.fAbsTarget := Spot_6X_StartTarget;
						点样轴7YDATE.fAbsTarget := Spot_7Y_Target;
						点样轴6XDATE.xMoveAbs := TRUE;
						点样轴7YDATE.xMoveAbs := TRUE;
						spot_band_step := 10;
					10:
						IF 点样轴6XDATE.bAbMoveDone AND 点样轴7YDATE.bAbMoveDone THEN
							点样轴6XDATE.xMoveAbs := FALSE;
							点样轴7YDATE.xMoveAbs := FALSE;
							IF %MW1300 = 0 AND NOT 泵站位符 THEN
								上样点样三通电池阀自动 := TRUE;
								上样吹气自动 := TRUE;
								泵站位符 := TRUE;
								转发转存 := Sampling_band_run_instruction;
								%MW1300 := LEN(STR:=转发转存);
								spot_band_step := 15;
							END_IF
						END_IF
					15:
						IF %MW1300 = 0 THEN
							泵站位符 := FALSE;
							IF Sampling_band_spot_speed > 0.0 THEN
								点样轴6XDATE.fVelocity := Sampling_band_spot_speed;
							END_IF
							点样轴6XDATE.fAbsTarget := Spot_6X_EndTarget;
							点样轴6XDATE.xMoveAbs := TRUE;
							spot_band_step := 20;
						END_IF
					20:
						IF 点样轴6XDATE.bAbMoveDone THEN
							点样轴6XDATE.xMoveAbs := FALSE;
							IF %MW1300 = 0 THEN
								泵站位符 := TRUE;
								转发转存 := Sampling_band_stop_instruction;
								%MW1300 := LEN(STR:=转发转存);
								spot_band_step := 25;
							END_IF
						END_IF
					25:
						IF %MW1300 = 0 THEN
							泵站位符 := FALSE;
							上样点样三通电池阀自动 := TRUE;
							上样吹气自动 := TRUE;
							spot_band_dry_count := 0;
							spot_band_step := 30;
						END_IF
					30:
							上样点样三通电池阀自动 := TRUE;
						上样吹气自动 := TRUE;
						IF Sampling_band_dry_speed > 0.0 THEN
							点样轴6XDATE.fVelocity := Sampling_band_dry_speed;
						END_IF
						点样轴6XDATE.fAbsTarget := Spot_6X_StartTarget;
						点样轴6XDATE.xMoveAbs := TRUE;
						spot_band_step := 40;
					40:
						IF 点样轴6XDATE.bAbMoveDone THEN
							点样轴6XDATE.xMoveAbs := FALSE;
								spot_band_step := 50;
						END_IF
					50:
							上样点样三通电池阀自动 := TRUE;
						上样吹气自动 := TRUE;
						IF Sampling_band_dry_speed > 0.0 THEN
							点样轴6XDATE.fVelocity := Sampling_band_dry_speed;
						END_IF
						点样轴6XDATE.fAbsTarget := Spot_6X_EndTarget;
						点样轴6XDATE.xMoveAbs := TRUE;
						spot_band_step := 60;
					60:
						IF 点样轴6XDATE.bAbMoveDone THEN
							点样轴6XDATE.xMoveAbs := FALSE;
							spot_band_dry_count := spot_band_dry_count + 1;
							IF spot_band_dry_count >= Sampling_band_dry_cycles THEN
								spot_band_step := 70;
							ELSE
							spot_band_step := 30;
							END_IF
						END_IF
					70:
							上样点样三通电池阀自动 := TRUE;
						上样吹气自动 := TRUE;
						点样轴6XDATE.fAbsTarget := HMI_点样轴6X.position[1];
						点样轴6XDATE.xMoveAbs := TRUE;
						spot_band_step := 80;
					80:
						IF 点样轴6XDATE.bAbMoveDone THEN
							点样轴6XDATE.xMoveAbs := FALSE;
							点样轴7YDATE.fAbsTarget := HMI_点样轴7Y.position[1];
							点样轴7YDATE.xMoveAbs := TRUE;
							spot_band_step := 90;
						END_IF
					90:
						IF 点样轴7YDATE.bAbMoveDone THEN
							点样轴7YDATE.xMoveAbs := FALSE;
							上样吹气自动 := FALSE;
							上样点样三通电池阀自动 := FALSE;
							IF spot_band_velocity_saved THEN
								点样轴6XDATE.fVelocity := spot_band_old_6x_velocity;
								spot_band_velocity_saved := FALSE;
							END_IF
							Sampling_Spray_sample_OK := TRUE;
							spot_band_step := 0;
							bActionDone := TRUE;
						END_IF
				END_CASE
		END_CASE
		IF bActionDone THEN
			bActionDone              := FALSE;
			Sampling_L2_CompletedSeq := Sampling_L2_AcceptedSeq;
			Sampling_L2_State        := 20;   (* DONE *)
		ELSIF bActionError THEN              (* 设备预条件未满足 -> 报错交上位机 *)
			bActionError             := FALSE;
			Sampling_L2_Retryable    := TRUE;
			Sampling_L2_CompletedSeq := Sampling_L2_AcceptedSeq;
			Sampling_L2_State        := 40;   (* ERROR; ErrorCode 由原子置 *)
		END_IF

	20, 30, 40, 50:  (* 终态: 等 Start 落沿或 Reset 回 IDLE *)
		IF (NOT Sampling_L2_Start) OR Sampling_L2_Reset THEN
			Sampling_L2_State := 0;
		END_IF
END_CASE

ACTION A50_absorb_吸收液体:
(* 吸收液体: Z回零->XY到坐标->Z下探->泵吸液循环->Z回零 (纯设备) *)
TON_0(IN:=吸收液体step=30, PT:=T#0.5S);
TON_1(IN:=NOT 点样气泡传感器, PT:=T#5S);
R_TRIG[10](CLK:=%MX2005.5);
// IF Sampling_X_coordinate>0 AND  Sampling_Y_coordinate>0  THEN
IF TRUE THEN
	CASE 吸收液体step OF
		0:
			上样轴5Z轴DATE.fAbsTarget:=0;
			上样轴5Z轴DATE.xMoveAbs:=TRUE;
			IF 上样轴5Z轴DATE.bAbMoveDone THEN
				上样轴5Z轴DATE.xMoveAbs:=FALSE;
// 				上样轴4X轴DATE.fAbsTarget:=HMI_上样轴4X轴.position[Sampling_X_coordinate];
// 				打样瓶上料轴3YDATE.fAbsTarget:=HMI_打样瓶上料轴3Y.position[Sampling_Y_coordinate];
				上样轴4X轴DATE.fAbsTarget:=Sampling_4X_Target;
				打样瓶上料轴3YDATE.fAbsTarget:=Sampling_3Y_Target;
				上样轴4X轴DATE.xMoveAbs:=TRUE;
				打样瓶上料轴3YDATE.xMoveAbs:=TRUE;
				吸收液体step:=10;
			END_IF
		10:
			IF 上样轴4X轴DATE.bAbMoveDone AND 打样瓶上料轴3YDATE.bAbMoveDone THEN
				上样轴4X轴DATE.xMoveAbs:=FALSE;
				打样瓶上料轴3YDATE.xMoveAbs:=FALSE;
				上样轴5Z轴DATE.fAbsTarget:=HMI_上样轴5Z轴.position[2];
				上样轴5Z轴DATE.xMoveAbs:=TRUE;
				吸收液体step:=20;
			END_IF
		20:
			IF 上样轴5Z轴DATE.bAbMoveDone THEN
				上样轴5Z轴DATE.xMoveAbs:=FALSE;
				A:=1;
				吸收液体step:=25;
			END_IF
		25:
			CASE A OF
				1,2:
					IF  %MW1300=0 AND NOT 泵站位符 THEN
						转发转存:=Sampling_sample_instructions[A];
						%MW1300:=LEN(STR:= 转发转存);
						泵站位符:=TRUE;
						吸收液体step:=30;
					END_IF
			END_CASE
		30:
			IF  %MW1300=0 AND TON_0.Q THEN
				转发转存:='/4Q$R';
				%MW1300:=LEN(STR:= 转发转存);
				IF R_TRIG[10].Q THEN
					泵站位符:=FALSE;
					A:=A+1;
					IF A>2 THEN
						A:=0;
						吸收液体step:=40;
					ELSE
						吸收液体step:=25;
					END_IF
				END_IF
			END_IF
		40:
			上样轴5Z轴DATE.fAbsTarget:=0;
			上样轴5Z轴DATE.xMoveAbs:=TRUE;
			IF 上样轴5Z轴DATE.bAbMoveDone THEN
				上样轴5Z轴DATE.xMoveAbs:=FALSE;
				Sampling_liquid_absorption:=TRUE;
				吸收液体step:=0;
				bActionDone:=TRUE;
			END_IF
	END_CASE
END_IF
END_ACTION

ACTION A31_放板移轴:
(* 放板移轴: 点样7Y轴到放板位 (上位机随后驱动机器人放板) *)
CASE 放硅胶板STEP OF
	0:
		点样轴7YDATE.fAbsTarget:=HMI_点样轴7Y.position[1];
		点样轴7YDATE.xMoveAbs:=TRUE;
		放硅胶板STEP:=10;
	10:
		IF 点样轴7YDATE.bAbMoveDone THEN
			点样轴7YDATE.xMoveAbs:=FALSE;
			放硅胶板STEP:=0;
			bActionDone:=TRUE;
		END_IF
END_CASE
END_ACTION

ACTION A40_prep_上样准备:
(* 上样准备: Z回零 + 注射泵准备指令循环 (纯设备) *)
TON[2](IN:=上样准备step=2,PT:=T#0.5S);
R_TRIG[3](CLK:=%MX2005.5);
CASE 上样准备step OF
	0:
		上样轴5Z轴DATE.fAbsTarget:=0;
		上样轴5Z轴DATE.xMoveAbs:=TRUE;
		IF 上样轴5Z轴DATE.bAbMoveDone THEN
			N:=1;
			上样轴5Z轴DATE.xMoveAbs:=FALSE ;
			上样准备step:=1;
		END_IF
	1:
		CASE N OF
			1,2:
				IF %MW1300=0 AND NOT 泵站位符 THEN
					泵站位符:=TRUE;
					转发转存:=Sampling_prep_instructions[N];
					%MW1300:=LEN(STR:= 转发转存);
					上样准备step:=2;
				END_IF
		END_CASE
	2:
		IF %MW1300=0 AND TON[2].Q THEN
		转发转存:='/4Q$R';
		%MW1300:=LEN(STR:= 转发转存);
		END_IF
		IF R_TRIG[3].Q THEN
			泵站位符:=FALSE;
			N:=N+1;
			IF N>2 THEN
				Sampling_preparation_OK:=TRUE;
				N:=0;
				上样准备step:=0;
				bActionDone:=TRUE;
			ELSE
				上样准备step:=1;
			END_IF
		END_IF
END_CASE
END_ACTION

ACTION A32_放板定位:
(* 放板定位: 上位机放板后定位夹紧 *)
上样定位自动:=TRUE;
Sampling_Place_materials_OK:=TRUE;
bActionDone:=TRUE;
END_ACTION

ACTION A20_clean_清洗:
(* 清洗: 伺服到清洗位 -> 注射泵清洗循环 Sampling_clean_count 次 (纯设备) *)
TON[1](IN:=清洗step=20,PT:=T#0.5S);
TON[6](IN:=清洗step=40,PT:=T#0.5S);
TON[8](IN:=清洗step=26,PT:=T#0.5S);
R_TRIG[2](CLK:=%MX2005.5);
R_TRIG[11](CLK:=%MX2005.5);
R_TRIG[12](CLK:=%MX2005.5);
CASE 清洗step OF
	0 :
		点样轴6XDATE.xMoveAbs:=FALSE;
		上样轴4X轴DATE.xMoveAbs:=FALSE;
		上样轴5Z轴DATE.xMoveAbs:=FALSE;
		清洗step:=5;
	5:
		点样轴6XDATE.fAbsTarget:=HMI_点样轴6X.position[1];
// 		上样轴4X轴DATE.fAbsTarget:=HMI_上样轴4X轴.position[9];
		上样轴4X轴DATE.fAbsTarget:=Sampling_4X_WashTarget;
		点样轴6XDATE.xMoveAbs:=TRUE;
		上样轴4X轴DATE.xMoveAbs:=TRUE;
		清洗计数:=0;
		清洗step:=6;
	6:
		IF 上样轴4X轴DATE.bAbMoveDone THEN
			上样轴4X轴DATE.xMoveAbs:=FALSE;
			上样轴5Z轴DATE.fAbsTarget:=HMI_上样轴5Z轴.position[1];
			上样轴5Z轴DATE.xMoveAbs:=TRUE;
			清洗step:=7;
		END_IF
	7:
		IF  上样轴5Z轴DATE.bAbMoveDone AND 点样轴6XDATE.bAbMoveDone THEN
			上样轴5Z轴DATE.xMoveAbs:=FALSE;
			点样轴6XDATE.xMoveAbs:=FALSE;
			IF Sampling_clean_count>0 THEN
				清洗step:=10;
			ELSE
				清洗step:=60;
			END_IF
		END_IF
	10:
		IF %MW1300=0 AND NOT 泵站位符 THEN
			泵站位符:=TRUE;
			转发转存:=Sampling_clean_instructions[1];
			%MW1300:=LEN(STR:= 转发转存);
			上样点样三通电池阀自动:=TRUE;
			清洗step:=20;
		END_IF
	20:
		IF %MW1300=0 AND TON[1].Q THEN
		转发转存:='/4Q$R';
		%MW1300:=LEN(STR:= 转发转存);
		END_IF
		IF R_TRIG[2].Q THEN
			上样点样三通电池阀自动:=FALSE;
			泵站位符:=FALSE;
			清洗step:=24;
		END_IF
	24:
		IF %MW1300=0 AND NOT 泵站位符 THEN
			泵站位符:=TRUE;
			转发转存:=Sampling_clean_instructions[1];
			%MW1300:=LEN(STR:= 转发转存);
			清洗step:=26;
		END_IF
	26:
		IF %MW1300=0 AND TON[8].Q THEN
		转发转存:='/4Q$R';
		%MW1300:=LEN(STR:= 转发转存);
		END_IF
		IF R_TRIG[11].Q THEN
			泵站位符:=FALSE;
			清洗step:=30;
		END_IF
	30:
		IF %MW1300=0 AND NOT 泵站位符 THEN
			泵站位符:=TRUE;
			转发转存:=Sampling_clean_instructions[2];
			%MW1300:=LEN(STR:= 转发转存);
			清洗step:=40;
		END_IF
	40:
		IF %MW1300=0 AND TON[6].Q THEN
		转发转存:='/4Q$R';
		%MW1300:=LEN(STR:= 转发转存);
		END_IF
		IF R_TRIG[12].Q THEN
			泵站位符:=FALSE;
			清洗step:=50;
		END_IF
	50:
		清洗计数:=清洗计数+1;
		IF  Sampling_clean_count> 清洗计数 THEN
			转发转存:='';
			%MW1300:=128;
			清洗step:=10;
		ELSIF  Sampling_clean_count<= 清洗计数 THEN
			转发转存:='';
			%MW1300:=128;
			清洗计数:=0;
			Sampling_Cleaning_OK:=TRUE;
			清洗step:=0;
			bActionDone:=TRUE;
		END_IF
		上样点样三通电池阀自动:=FALSE;
	60:
		Sampling_Cleaning_OK:=TRUE;
		清洗step:=0;
		bActionDone:=TRUE;
END_CASE
END_ACTION

ACTION A10_init_初始化:
(* 初始化: 复位阀/伺服回零 + 注射泵初始化 (已删机器人握手位复位) *)
CASE 初始化step OF
	0 :
		上样定位手动:=FALSE;
		上样定位自动:=FALSE;
		上样点样三通电池阀手动:=FALSE;
		上样点样三通电池阀自动:=FALSE;
		上样吹气手动:=FALSE;
		上样吹气自动:=FALSE;
		打样瓶上料轴3YDATE.fAbsTarget:=0;
		点样轴6XDATE.fAbsTarget:=0;
		点样轴7YDATE.fAbsTarget:=0;
		上样轴4X轴DATE.fAbsTarget:=0;
		上样轴5Z轴DATE.fAbsTarget:=0;
		点样轴7YDATE.xMoveAbs:=FALSE;
		点样轴6XDATE.xMoveAbs:=FALSE;
		上样轴5Z轴DATE.xMoveAbs:=FALSE;
		上样轴4X轴DATE.xMoveAbs:=FALSE;
		打样瓶上料轴3YDATE.xMoveAbs:=FALSE;
		Sampling_Spray_sample_OK:=FALSE;
		Sampling_liquid_absorption:=FALSE;
		Sampling_preparation_OK:=FALSE;
		大真空泵站位[11]:=FALSE;
		清洗计数:=0;
		清洗step:=0;
		放硅胶板STEP:=0;
		上样准备step:=0;
		吸收液体step:=0;
		点样step:=0;
		初始化step:=5;
	5:
		上样轴5Z轴DATE.fAbsTarget:=0;
		上样轴5Z轴DATE.xMoveAbs:=TRUE;
		IF 上样轴5Z轴DATE.bAbMoveDone THEN
			点样轴7YDATE.fAbsTarget:=0  ;
			点样轴6XDATE.fAbsTarget:=0  ;
			上样轴4X轴DATE.fAbsTarget:=0;
			上样轴4X轴DATE.xMoveAbs:=TRUE;
			点样轴7YDATE.xMoveAbs:=TRUE;
			点样轴6XDATE.xMoveAbs:=TRUE;
			初始化step:=6;
		END_IF
	6:
		IF 上样轴4X轴DATE.bAbMoveDone AND 上样轴5Z轴DATE.bAbMoveDone AND 点样轴6XDATE.bAbMoveDone AND 点样轴7YDATE.bAbMoveDone THEN
			初始化step:=10;
			上样轴4X轴DATE.xMoveAbs:=FALSE;
			点样轴7YDATE.xMoveAbs:=FALSE;
			上样轴5Z轴DATE.xMoveAbs:=FALSE;
			点样轴6XDATE.xMoveAbs:=FALSE;
		END_IF
	10:
		IF %MW1300=0 AND NOT 泵站位符 THEN
			泵站位符:=TRUE;
			转发转存:='/4Z0,1,1R$R';
			%MW1300:=LEN(STR:= 转发转存);
			初始化STEP:=20;
		END_IF
	20:
		IF %MW1300=0 THEN
			转发转存:='/4Q$R';
			%MW1300:=LEN(STR:= 转发转存);
		END_IF
		R_TRIG[1](CLK:=%MX2005.5);
		IF R_TRIG[1].Q THEN
			泵站位符:=FALSE;
			初始化STEP:=30;
		END_IF
	30:
		Sampling_initialization_OK:=TRUE;
		初始化step:=0;
		bActionDone:=TRUE;
END_CASE
END_ACTION

ACTION A60_spray_点样:
(* 点样: 伺服点样序列 + 注射泵点样 (已删尾部 允许取硅胶板 机器人握手) *)
TON[4](IN:=点样step=20,PT:=T#0.5S);
TON[5](IN:=点样气泡传感器,PT:=T#5S);
TON[7](IN:=点样step=10,PT:=T#0.5S);
R_TRIG[10](CLK:=%MX2005.5);
CASE 点样step OF
	0:
		点样轴6XDATE.xMoveAbs:=FALSE;
		点样轴7YDATE.xMoveAbs:=FALSE;
		点样step:=1;
	1:
// 		点样轴6XDATE.fAbsTarget:=HMI_点样轴6X.position[2];
		点样轴6XDATE.fAbsTarget:=Spot_6X_StartTarget;
// 		点样轴7YDATE.fAbsTarget:=HMI_点样轴7Y.position[2];
		点样轴7YDATE.fAbsTarget:=Spot_7Y_Target;
		点样轴6XDATE.xMoveAbs:=TRUE;
		点样轴7YDATE.xMoveAbs:=TRUE;
		点样step:=5;
	5:
		IF 点样轴6XDATE.bAbMoveDone AND 点样轴7YDATE.bAbMoveDone THEN
			点样轴6XDATE.xMoveAbs:=FALSE;
			点样轴7YDATE.xMoveAbs:=FALSE;
			IF  %MW1300=0 AND NOT 泵站位符 THEN
				泵站位符:=TRUE;
				转发转存:=Sampling_dispense_instructions[1];
				%MW1300:=LEN(STR:= 转发转存);
				上样点样三通电池阀自动:=TRUE;
				点样step:=10;
			END_IF
		END_IF
	10:
		IF  %MW1300=0 AND TON[7].Q THEN
				转发转存:='/4Q$R';
				%MW1300:=LEN(STR:= 转发转存);
				IF R_TRIG[10].Q THEN
					泵站位符:=FALSE;
					点样step:=15;
				END_IF
		END_IF
	15:
		IF  %MW1300=0 AND NOT 泵站位符 THEN
			上样吹气自动:=TRUE;
			泵站位符:=TRUE;
			转发转存:=Sampling_dispense_instructions[2];
			%MW1300:=LEN(STR:= 转发转存);
// 			点样轴6XDATE.fAbsTarget:=HMI_点样轴6X.position[3];
			点样轴6XDATE.fAbsTarget:=Spot_6X_EndTarget;
			点样轴6XDATE.xMoveAbs:=TRUE;
			点样step:=20;
		END_IF
	20:
		IF  %MW1300=0 AND TON[4].Q THEN
				转发转存:='/4Q$R';
				%MW1300:=LEN(STR:= 转发转存);
				IF R_TRIG[10].Q THEN
					泵站位符:=FALSE;
					上样点样三通电池阀自动:=FALSE;
					上样吹气自动:=FALSE;
				END_IF
		END_IF
		CASE 打样伺服移动step OF
			0:
				IF 点样轴6XDATE.bAbMoveDone THEN
					点样轴6XDATE.xMoveAbs:=FALSE;
					IF 泵站位符 THEN
						打样伺服移动step:=10;
					ELSE
						点样step:=30;
					END_IF
				END_IF
			10:
// 				点样轴6XDATE.fAbsTarget:=HMI_点样轴6X.position[2];
				点样轴6XDATE.fAbsTarget:=Spot_6X_StartTarget;
				点样轴6XDATE.xMoveAbs:=TRUE;
				打样伺服移动step:=20;
			20:
				IF 点样轴6XDATE.bAbMoveDone THEN
					点样轴6XDATE.xMoveAbs:=FALSE;
					打样伺服移动step:=30;
				END_IF
			30:
// 				点样轴6XDATE.fAbsTarget:=HMI_点样轴6X.position[3];
				点样轴6XDATE.fAbsTarget:=Spot_6X_EndTarget;
				点样轴6XDATE.xMoveAbs:=TRUE;
				打样伺服移动step:=0;
		END_CASE
	30:
		点样轴6XDATE.fAbsTarget:=HMI_点样轴6X.position[1];
		点样轴6XDATE.xMoveAbs:=TRUE;
		IF 点样轴6XDATE.bAbMoveDone THEN
			点样轴7YDATE.fAbsTarget:=HMI_点样轴7Y.position[1];
			点样轴7YDATE.xMoveAbs:=TRUE;
			点样step:=40;
		END_IF
	40:
		IF 点样轴7YDATE.bAbMoveDone  THEN
			点样轴6XDATE.xMoveAbs:=FALSE;
			点样轴7YDATE.xMoveAbs:=FALSE;
			上样定位自动:=FALSE;
			Sampling_Spray_sample_OK:=TRUE;
			点样step:=0;
			bActionDone:=TRUE;
		END_IF
END_CASE
END_ACTION

ACTION A61_喷涂移轴:
CASE 喷涂移轴step OF
					0:
						点样轴7YDATE.fAbsTarget := HMI_点样轴7Y.position[2];
						点样轴7YDATE.xMoveAbs := TRUE;
						喷涂移轴step := 10;
					10:
						IF 点样轴7YDATE.bAbMoveDone THEN
							点样轴7YDATE.xMoveAbs := FALSE;
							喷涂移轴step := 0;
							bActionDone := TRUE;
						END_IF
				END_CASE
END_ACTION

END_PROGRAM

// Device/Application/50_action/Collect_L2
PROGRAM Collect_L2
VAR
	初始化STEP: INT;
	准备step: INT;
	收集step: INT;
	搬运step: INT;
	泵初始化完成: BOOL;
	bActionDone: BOOL;
	bActionError: BOOL;
	L2_StartTrig: R_TRIG;
	R_TRIG: ARRAY[1..5] OF R_TRIG;
	ton: ARRAY[1..10] OF TON;
	TON_0: TON;
END_VAR

(* 收集工位 L2 统一动作派发器
   功能:
       按 Collect_L2_ActionCode 把上位机请求派发到设备原子动作 (纯设备, 不含机器人握手).
   协议:
       Collect_L2_Start 上升沿接受请求 -> RUNNING 每周期调用对应原子 -> 原子置 bActionDone -> DONE.
   动作码:
       10 init 初始化 / 21 夹持夹紧 / 22 伸缩伸出 / 23 缩回升降下压
       30 collect 收集 / 41 复位伸出 / 42 伸缩缩回 / 43 松夹持
   参数:
       无, 经 Collect_L2_* 反馈. *)
L2_StartTrig(CLK := Collect_L2_Start);

CASE Collect_L2_State OF
	0:  (* IDLE *)
		Collect_L2_Step := 0;
		IF L2_StartTrig.Q THEN
			Collect_L2_AcceptedSeq := Collect_L2_RequestSeq;
			Collect_L2_ActiveCode  := Collect_L2_ActionCode;
			Collect_L2_ErrorCode   := 0;
			Collect_L2_Retryable   := FALSE;
			bActionDone            := FALSE;
			bActionError           := FALSE;
			初始化STEP := 0;
			准备step   := 0;
			收集step   := 0;
			搬运step   := 0;
			CASE Collect_L2_ActionCode OF
				10, 21, 22, 23, 24, 30, 41, 42, 43:
					Collect_L2_SafeState := 0;
					Collect_L2_State     := 10;   (* RUNNING *)
			ELSE
				Collect_L2_ErrorCode    := 101;  (* 未知动作码 *)
				Collect_L2_Retryable    := TRUE;
				Collect_L2_CompletedSeq := Collect_L2_AcceptedSeq;
				Collect_L2_State        := 30;   (* REJECTED *)
			END_CASE
		END_IF

	10: (* RUNNING *)
		IF Collect_L2_Reset THEN Collect_L2_State := 0; RETURN; END_IF   (* RUNNING 中 RESET: 中止挂死动作 *)
		CASE Collect_L2_ActiveCode OF
			10: A10_init_初始化();
			21: A21_夹持夹紧();
			22: A22_伸缩伸出();
			23: A23_缩回升降下压();
			24: 溶液收集瓶定位自动:=Collect_BottleLocate_Target; bActionDone:=TRUE;
			30: A30_collect_收集();
			41: A41_复位伸出();
			42: A42_伸缩缩回();
			43: A43_松夹持();
		END_CASE
		IF bActionDone THEN
			bActionDone             := FALSE;
			Collect_L2_CompletedSeq := Collect_L2_AcceptedSeq;
			Collect_L2_State        := 20;   (* DONE *)
		ELSIF bActionError THEN              (* 设备预条件未满足 -> 报错交上位机 *)
			bActionError            := FALSE;
			Collect_L2_Retryable    := TRUE;
			Collect_L2_CompletedSeq := Collect_L2_AcceptedSeq;
			Collect_L2_State        := 40;   (* ERROR; ErrorCode 由原子置 *)
		END_IF

	20, 30, 40, 50:  (* 终态: 等 Start 落沿或 Reset 回 IDLE *)
		IF (NOT Collect_L2_Start) OR Collect_L2_Reset THEN
			Collect_L2_State := 0;
		END_IF
END_CASE

ACTION A23_缩回升降下压:
(* 缩回 -> 升降上升 -> 下压 (上位机已先驱动机器人放收集瓶)
   缺瓶处理: 原 A10 "缺瓶重试" 改为报错交上位机 (ErrorCode 201), 由上位机重放瓶后重调 *)
CASE 准备step OF
	0:
		收集伸缩气缸自动:=FALSE;
		准备step:=10;
	10:
		IF 收集平台推出气缸原点 AND 收集平台瓶子有无传感器 THEN
			收集升降气缸自动:=TRUE;
			准备step:=20;
		ELSIF 收集平台推出气缸原点 AND NOT 收集平台瓶子有无传感器 THEN
			准备step:=0;
			Collect_L2_ErrorCode:=201;   (* 缺瓶: 上位机放瓶后传感器未检到 *)
			bActionError:=TRUE;
		END_IF
	20:
		IF 收集平台升降气缸动点 THEN
			收集下压气缸自动:=TRUE;
			准备step:=0;
			bActionDone:=TRUE;
		END_IF
END_CASE
END_ACTION

ACTION A22_伸缩伸出:
(* 伸缩气缸伸出到放瓶位 *)
CASE 准备step OF
	0:
		IF 收集平台推出气缸原点 AND NOT 收集平台瓶子有无传感器 THEN
			收集伸缩气缸自动:=TRUE;
			准备step:=10;
		END_IF
	10:
		IF 收集平台推出气缸动点 THEN
			准备step:=0;
			bActionDone:=TRUE;
		END_IF
END_CASE
END_ACTION

ACTION A21_夹持夹紧:
(* 夹持气缸夹紧 (上位机已先驱动机器人放收集器) *)
CASE 准备step OF
	0:
		收集夹持气缸自动:=TRUE;
		准备step:=10;
	10:
		IF 收集平台夹持气缸动点 THEN
			准备step:=0;
			bActionDone:=TRUE;
		END_IF
END_CASE
END_ACTION

ACTION A30_collect_收集:
(* 收集: 进液 -> 注射泵转发 -> 排液/正压循环 collect_count 次 (纯设备, 不变) *)
ton[1](IN:=收集step=10, PT:=T#0.5S);
ton[2](IN:=收集step=30, PT:=T#10S);
R_TRIG[5](CLK := %MX2005.5);
CASE 收集step OF
	0:
		IF collect_forward_instructions<>'' THEN
			收集进液自动:=TRUE;
		END_IF
		IF %MW1300=0 AND 泵站位符=FALSE THEN
			转发转存:=collect_forward_instructions;
			%MW1300:=LEN(STR:= 转发转存);
			泵站位符:=TRUE;
			收集step:=10;
		END_IF
	10:
		IF %MW1300=0 AND ton[1].Q THEN
			转发转存:='/3Q$R';
			%MW1300:=LEN(STR:= 转发转存);
		END_IF
		IF R_TRIG[5].Q THEN
			泵站位符:=FALSE;
			收集step:=20;
		END_IF
	20:
		转发转存:='';
		%MW1300:=128;
		收集进液自动:=FALSE;
		收集排液自动:=TRUE;
		收集正压排液自动:=TRUE;
		收集计数:=收集计数+1;
		收集step:=30;
	30:
		TON_0(IN:=ton[2].Q, PT:=T#5S);   (* 排液计时后再沉淀, 沉淀完成才判定, 杜绝误回 step0 *)
		IF TON_0.Q THEN
			IF 收集计数>=collect_count THEN
				收集计数:=0;
				收集step:=40;
			ELSE
				收集排液自动:=FALSE;
				收集正压排液自动:=FALSE;
				收集step:=0;
			END_IF
		END_IF
	40:
		收集排液自动:=FALSE;
		收集正压排液自动:=FALSE;
		收集step:=0;
		bActionDone:=TRUE;
END_CASE
END_ACTION

ACTION A10_init_初始化:
(* 初始化: 复位气缸/电磁阀 + 注射泵初始化 (已删机器人握手位复位)
   完成条件: 四气缸回原点 AND 泵初始化完成 *)
R_TRIG[1](CLK := %MX2005.5);   (* 泵空闲上升沿 *)
CASE 初始化STEP OF
	0:
		溶液收集瓶定位自动:=FALSE;
		收集下压气缸手动:=FALSE; 收集下压气缸自动:=FALSE;
		收集夹持气缸手动:=FALSE; 收集夹持气缸自动:=FALSE;
		收集升降气缸手动:=FALSE; 收集升降气缸自动:=FALSE;
		收集伸缩气缸手动:=FALSE; 收集伸缩气缸自动:=FALSE;
		收集进液手动:=FALSE; 收集进液自动:=FALSE;
		收集排液手动:=FALSE; 收集排液自动:=FALSE;
		收集正压排液手动:=FALSE; 收集正压排液自动:=FALSE;
		溶液收集瓶定位手动:=FALSE;
		IF %MW1300=0 AND NOT 泵站位符 THEN
			泵站位符:=TRUE;
			转发转存:='/3Z0,2,2R$R';             (* 泵初始化指令 *)
			%MW1300:=LEN(STR:= 转发转存);
			初始化STEP:=10;
		END_IF
	10:
		IF %MW1300=0 THEN
			转发转存:='/3Q$R';                   (* 查询泵状态 *)
			%MW1300:=LEN(STR:= 转发转存);
		END_IF
		IF R_TRIG[1].Q THEN
			泵站位符:=FALSE;
			泵初始化完成:=TRUE;
			初始化STEP:=20;
		END_IF
	20:
		IF 收集平台下压气缸原点 AND 收集平台夹持气缸原点
		   AND 收集平台升降气缸原点 AND 收集平台推出气缸原点
		   AND 泵初始化完成 THEN
			泵初始化完成:=FALSE;
			初始化STEP:=0;
			bActionDone:=TRUE;
		END_IF
END_CASE
END_ACTION

ACTION A42_伸缩缩回:
(* 搬运段2: 伸缩缩回 (上位机已先驱动机器人取瓶到暂存) *)
CASE 搬运step OF
	0:
		收集伸缩气缸自动:=FALSE;
		搬运step:=10;
	10:
		IF 收集平台推出气缸原点 THEN
			搬运step:=0;
			bActionDone:=TRUE;
		END_IF
END_CASE
END_ACTION

ACTION A41_复位伸出:
(* 搬运段1: 复位下压/升降 -> 伸缩伸出到取瓶位 *)
CASE 搬运step OF
	0:
		收集下压气缸自动:=FALSE;
		搬运step:=5;
	5:
		IF 收集平台下压气缸原点 THEN
			收集升降气缸自动:=FALSE;
			搬运step:=10;
		END_IF
	10:
		IF 收集平台升降气缸原点 THEN
			收集伸缩气缸自动:=TRUE;
			搬运step:=20;
		END_IF
	20:
		IF 收集平台推出气缸动点 THEN
			搬运step:=0;
			bActionDone:=TRUE;
		END_IF
END_CASE
END_ACTION

ACTION A43_松夹持:
(* 搬运段3: 松夹持 (上位机已先驱动机器人到收集器位) *)
CASE 搬运step OF
	0:
		收集夹持气缸自动:=FALSE;
		搬运step:=10;
	10:
		IF 收集平台夹持气缸原点 THEN
			搬运step:=0;
			bActionDone:=TRUE;
		END_IF
END_CASE
END_ACTION

END_PROGRAM

// Device/Application/50_action/Develop_L2
PROGRAM Develop_L2
VAR
	初始化step: INT;
	清洗STEP: INT;
	润洗展缸STEP: INT;
	上液step: INT;
	放硅胶板step: INT;
	润洗计数: INT;
	上液计数: INT;
	泵初始化完成: BOOL;
	bActionDone: BOOL;
	bActionError: BOOL;
	TON_0: TON;
	TON_1: TON;
	TON_2: TON;
	DrainTank: INT;
	L2_StartTrig: R_TRIG;
	R_TRIG: ARRAY[1..10] OF R_TRIG;
	TON: ARRAY[1..10] OF TON;
END_VAR

(* Develop 工位 L2 统一动作派发器
   按 Develop_L2_ActionCode 派发到纯设备原子动作 (不含机器人/相机/CNC 握手).
   Start 上升沿接受请求 -> RUNNING 每周期调用对应原子 -> bActionDone=DONE / bActionError=ERROR. *)
L2_StartTrig(CLK := Develop_L2_Start);

CASE Develop_L2_State OF
	0:  (* IDLE *)
		Develop_L2_Step := 0;
		IF L2_StartTrig.Q THEN
			Develop_L2_AcceptedSeq := Develop_L2_RequestSeq;
			Develop_L2_ActiveCode  := Develop_L2_ActionCode;
			Develop_L2_ErrorCode   := 0;
			Develop_L2_Retryable   := FALSE;
			bActionDone  := FALSE;
			bActionError := FALSE;
			初始化step := 0;
			清洗STEP := 0;
			润洗展缸STEP := 0;
			上液step := 0;
			放硅胶板step := 0;
			DrainTank := Expand_Target_Tank;
			IF (DrainTank < 1) OR (DrainTank > 8) THEN
				Develop_L2_ErrorCode    := 102;  (* target tank out of range *)
				Develop_L2_Retryable    := TRUE;
				Develop_L2_CompletedSeq := Develop_L2_AcceptedSeq;
				Develop_L2_State        := 30;   (* REJECTED *)
			ELSE
				Expand_Group  := (DrainTank - 1) / 4 + 1;
				Expand_Number := (DrainTank - 1) MOD 4 + 1;
				CASE Develop_L2_ActionCode OF
					10, 20, 21, 22, 26, 31, 32:
						Develop_L2_SafeState := 0;
						Develop_L2_State     := 10;   (* RUNNING *)
					50:
						IF Tank_State[DrainTank] = 40 THEN
							Tank_Drain_Enable[DrainTank] := TRUE;
							Develop_L2_SafeState := 0;
							Develop_L2_State     := 10;   (* RUNNING *)
						ELSIF Tank_State[DrainTank] = 99 THEN
							Develop_L2_SafeState := 10;
							Develop_L2_State     := 10;   (* RUNNING; idempotent done path *)
						ELSE
							Develop_L2_ErrorCode    := 501;  (* tank is not Developing/Done *)
							Develop_L2_Retryable    := TRUE;
							Develop_L2_CompletedSeq := Develop_L2_AcceptedSeq;
							Develop_L2_State        := 30;   (* REJECTED *)
						END_IF
					51:
						IF (Tank_State[DrainTank] = 99) OR (Tank_State[DrainTank] = 0) THEN
							Develop_L2_SafeState := 10;
							Develop_L2_State     := 10;   (* RUNNING; release is scan-local *)
						ELSE
							Develop_L2_ErrorCode    := 511;  (* only Done/Idle tank can be released *)
							Develop_L2_Retryable    := TRUE;
							Develop_L2_CompletedSeq := Develop_L2_AcceptedSeq;
							Develop_L2_State        := 30;   (* REJECTED *)
						END_IF
				ELSE
					Develop_L2_ErrorCode    := 101;  (* unknown action code *)
					Develop_L2_Retryable    := TRUE;
					Develop_L2_CompletedSeq := Develop_L2_AcceptedSeq;
					Develop_L2_State        := 30;   (* REJECTED *)
				END_CASE
			END_IF
		END_IF

	10: (* RUNNING *)
		IF Develop_L2_Reset THEN
			IF Develop_L2_ActiveCode = 50 THEN
				Tank_Drain_Enable[DrainTank] := FALSE;
			END_IF
			Develop_L2_State := 0;
			RETURN;
		END_IF   (* RUNNING reset aborts stuck action *)
		CASE Develop_L2_ActiveCode OF
			10: A10_init_初始化();
			20: A20_pipeline_清洗管路();
			21: A21_rinse_润洗展缸();
			26: A26_rinse_suction();
			22: A22_up_liquid_上液();
			31: A31_放板缸回原点();
			32: A32_放板缸到动点();
			50:
				Develop_L2_Step := Tank_State[DrainTank];
				IF Tank_State[DrainTank] = 90 THEN
					Develop_L2_ErrorCode := 502;  (* drain FSM error *)
					bActionError := TRUE;
				ELSIF (Tank_State[DrainTank] = 99) OR Tank_Drain_Done[DrainTank] THEN
					Develop_L2_SafeState := 10;
					bActionDone := TRUE;
				END_IF
			51:
				Develop_L2_Step := Tank_State[DrainTank];
				IF (Tank_State[DrainTank] = 99) OR (Tank_State[DrainTank] = 0) THEN
					Tank_Drain_Enable[DrainTank] := FALSE;
					Tank_Drain_Done[DrainTank] := FALSE;
					Tank_State[DrainTank] := 0;
					Develop_L2_SafeState := 10;
					bActionDone := TRUE;
				ELSE
					Develop_L2_ErrorCode := 511;
					bActionError := TRUE;
				END_IF
		END_CASE
		IF bActionDone THEN
			bActionDone              := FALSE;
			Develop_L2_CompletedSeq := Develop_L2_AcceptedSeq;
			Develop_L2_State        := 20;   (* DONE *)
		ELSIF bActionError THEN              (* 设备预条件未满足 -> 报错交上位机 *)
			bActionError             := FALSE;
			Develop_L2_Retryable    := TRUE;
			Develop_L2_CompletedSeq := Develop_L2_AcceptedSeq;
			Develop_L2_State        := 40;   (* ERROR; ErrorCode 由原子置 *)
		END_IF

	20, 30, 40, 50:  (* terminal: wait Start falling edge or Reset *)
		IF (NOT Develop_L2_Start) OR Develop_L2_Reset THEN
			IF Develop_L2_ActiveCode = 50 THEN  (* terminal drain cleanup *)
				Tank_Drain_Enable[DrainTank] := FALSE;
			END_IF
			Develop_L2_State := 0;
		END_IF
END_CASE

ACTION A31_放板缸回原点:
(* 放板-缸回原点 (上位机随后驱动机器人放板); 删原机器人到位/允许握手 *)
CASE Expand_Group OF
	1:
		CASE Expand_Number OF
			1:
				展缸1气缸1自动:=FALSE;
				IF 展缸1气缸1原点 THEN bActionDone:=TRUE; END_IF
			2:
				展缸1气缸2自动:=FALSE;
				IF 展缸1气缸2原点 THEN bActionDone:=TRUE; END_IF
			3:
				展缸1气缸3自动:=FALSE;
				IF 展缸1气缸3原点 THEN bActionDone:=TRUE; END_IF
			4:
				展缸1气缸4自动:=FALSE;
				IF 展缸1气缸4原点 THEN bActionDone:=TRUE; END_IF
		END_CASE
	2:
		CASE Expand_Number OF
			1:
				展缸2气缸1自动:=FALSE;
				IF 展缸2气缸1原点 THEN bActionDone:=TRUE; END_IF
			2:
				展缸2气缸2自动:=FALSE;
				IF 展缸2气缸2原点 THEN bActionDone:=TRUE; END_IF
			3:
				展缸2气缸3自动:=FALSE;
				IF 展缸2气缸3原点 THEN bActionDone:=TRUE; END_IF
			4:
				展缸2气缸4自动:=FALSE;
				IF 展缸2气缸4原点 THEN bActionDone:=TRUE; END_IF
		END_CASE
END_CASE
END_ACTION

ACTION A21_rinse_润洗展缸:
TON[1](IN:=润洗展缸STEP=15,PT:=T#0.1S);
TON_1(IN:= 润洗展缸STEP=20  , PT:=T#5S , Q=> , ET=> );
TON_2(IN:=润洗展缸STEP=30, PT:=T#3S, Q=> , ET=> );
TON[4](IN:=润洗展缸STEP=40,PT:=T#30S);
TON[10](IN:=(Expand_Group=1 AND  展缸1溶剂废液检测传感器) OR (Expand_Group=2 AND  展缸2溶剂废液检测传感器),PT:=T#10S);
R_TRIG[3](CLK:=%MX2005.5 , Q=> );  //泵空闲中



CASE 润洗展缸STEP OF
	0 :
		润洗计数:=0;
		CASE Expand_Group OF
			1:
				CASE Expand_Number OF
					1:
						展缸1进液电池阀1自动:=TRUE;
						展缸1排液电池阀1自动:=TRUE;
						展缸1气缸1自动:=TRUE;
						润洗展缸STEP:=10;
					2:
						展缸1进液电池阀2自动:=TRUE;
						展缸1排液电池阀2自动:=TRUE;
						展缸1气缸2自动:=TRUE;
						润洗展缸STEP:=10;
					3:
						展缸1进液电池阀3自动:=TRUE;
						展缸1排液电池阀3自动:=TRUE;
						展缸1气缸3自动:=TRUE;
						润洗展缸STEP:=10;
					4:
						展缸1进液电池阀4自动:=TRUE;
						展缸1排液电池阀4自动:=TRUE;
						展缸1气缸4自动:=TRUE;
						润洗展缸STEP:=10;
				END_CASE
			
			2:
				CASE Expand_Number OF
					1:
						展缸2进液电池阀1自动:=TRUE;
						展缸2排液电池阀1自动:=TRUE;
						展缸2气缸1自动:=TRUE;
						润洗展缸STEP:=10;
					2:
						展缸2进液电池阀2自动:=TRUE;
						展缸2排液电池阀2自动:=TRUE;
						展缸2气缸2自动:=TRUE;
						润洗展缸STEP:=10;
					3:
						展缸2进液电池阀3自动:=TRUE;
						展缸2排液电池阀3自动:=TRUE;
						展缸2气缸3自动:=TRUE;
						润洗展缸STEP:=10;
					4:
						展缸2进液电池阀4自动:=TRUE;
						展缸2排液电池阀4自动:=TRUE;
						展缸2气缸4自动:=TRUE;
						润洗展缸STEP:=10;
				END_CASE
		END_CASE
	10:		
		IF %MW1300=0 AND 泵站位符=FALSE  THEN
			转发转存:=Expand_forward_instructions;   
			%MW1300:=LEN(STR:= 转发转存);   //发送字节数
			泵站位符:=TRUE;
			润洗展缸STEP:=15;
		END_IF
	15:
		
		IF %MW1300=0 AND TON[1].Q THEN
			CASE Expand_Group OF
				1:
					转发转存:='/1Q$R';           //查询泵状态指令
				2:
					转发转存:='/2Q$R';           //查询泵状态指令
			END_CASE
			%MW1300:=LEN(STR:= 转发转存);
		END_IF
		
		IF R_TRIG[3].Q THEN
			泵站位符:=FALSE;
			润洗计数:=润洗计数+1;
			IF 润洗计数>=Expand_rinse_count THEN
				润洗计数:=0;
				润洗展缸STEP:=20;
			ELSE
				润洗展缸STEP:=10;
			END_IF
			
		END_IF
		
	20:
		//TON_1(IN:= TRUE  , PT:=T#5S , Q=> , ET=> );
		IF TON_1.Q THEN
			转发转存:='';
			%MW1300:=128;
			Expand_Group_clean_OK:=TRUE; bActionDone:=TRUE;
			润洗展缸STEP:=0;
		END_IF
END_CASE
END_ACTION

ACTION A20_pipeline_清洗管路:
TON[2](IN:=清洗STEP=10,PT:=T#1S);
TON_0(IN:=清洗STEP=20, PT:=T#3S , Q=> , ET=> );
R_TRIG[5](CLK:=%MX2005.5 , Q=> );  //泵空闲中
CASE 清洗STEP OF
	0 :
		IF %MW1300=0 AND 泵站位符=FALSE  THEN
			转发转存:=Expand_forward_instructions; 
			%MW1300:=LEN(STR:= 转发转存);   //发送字节数
			泵站位符:=TRUE;
			清洗STEP:=10;
		END_IF
	10:
		//TON[2](IN:=TRUE,PT:=T#1S);
		IF %MW1300=0 AND TON[2].Q THEN
			CASE Expand_Group OF
				1:
					转发转存:='/1Q$R';          //查询泵状态指令
				2:
					转发转存:='/2Q$R';          //查询泵状态指令
			END_CASE
			%MW1300:=LEN(STR:= 转发转存);
		END_IF
		
		
		IF R_TRIG[5].Q THEN
			泵站位符:=FALSE;
			清洗STEP:=20;
		END_IF
	20:
		
		IF TON_0.Q THEN
			转发转存:='';
			%MW1300:=128;
			Expand_Group_clean_OK:=TRUE; bActionDone:=TRUE;
			清洗STEP:=0;
		END_IF

		
END_CASE
END_ACTION

ACTION A32_放板缸到动点:
(* 放板-缸到动点 (上位机已驱动机器人放完板) *)
CASE Expand_Group OF
	1:
		CASE Expand_Number OF
			1:
				展缸1气缸1自动:=TRUE;
				IF 展缸1气缸1动点 THEN bActionDone:=TRUE; END_IF
			2:
				展缸1气缸2自动:=TRUE;
				IF 展缸1气缸2动点 THEN bActionDone:=TRUE; END_IF
			3:
				展缸1气缸3自动:=TRUE;
				IF 展缸1气缸3动点 THEN bActionDone:=TRUE; END_IF
			4:
				展缸1气缸4自动:=TRUE;
				IF 展缸1气缸4动点 THEN bActionDone:=TRUE; END_IF
		END_CASE
	2:
		CASE Expand_Number OF
			1:
				展缸2气缸1自动:=TRUE;
				IF 展缸2气缸1动点 THEN bActionDone:=TRUE; END_IF
			2:
				展缸2气缸2自动:=TRUE;
				IF 展缸2气缸2动点 THEN bActionDone:=TRUE; END_IF
			3:
				展缸2气缸3自动:=TRUE;
				IF 展缸2气缸3动点 THEN bActionDone:=TRUE; END_IF
			4:
				展缸2气缸4自动:=TRUE;
				IF 展缸2气缸4动点 THEN bActionDone:=TRUE; END_IF
		END_CASE
END_CASE
END_ACTION

ACTION A22_up_liquid_上液:
R_TRIG[6](CLK:=%MX2005.5 , Q=> );  //泵空闲中
TON[9](IN:=上液step=20,PT:=T#0.5S,);
IF Expand_Group>0 AND Expand_Number>0 THEN
	CASE 上液step OF
		0:
			CASE Expand_Group OF
				1:
					CASE Expand_Number OF
						1:
							展缸1进液电池阀1自动:=TRUE;
							上液step:=10;
						2:
							展缸1进液电池阀2自动:=TRUE;
							上液step:=10;
						3:
							展缸1进液电池阀3自动:=TRUE;
							上液step:=10;
						4:
							展缸1进液电池阀4自动:=TRUE;
							上液step:=10;
					END_CASE
				2:
					CASE Expand_Number OF
						1:
							展缸2进液电池阀1自动:=TRUE;
							上液step:=10;
						2:
							展缸2进液电池阀2自动:=TRUE;
							上液step:=10;
						3:
							展缸2进液电池阀3自动:=TRUE;
							上液step:=10;
						4:
							展缸2进液电池阀4自动:=TRUE;
							上液step:=10;
					END_CASE
			END_CASE
		10:
			IF %MW1300=0 AND 泵站位符=FALSE  THEN
				转发转存:=Expand_forward_instructions; 
				%MW1300:=LEN(STR:= 转发转存);   //发送字节数
				泵站位符:=TRUE;
				上液step:=20;
			END_IF
		20:
		
			IF %MW1300=0 AND TON[9].Q  THEN
				CASE Expand_Group OF
					 1:
						 转发转存:='/1Q$R';          //查询泵状态指令
					 2:
						 转发转存:='/2Q$R';          //查询泵状态指令
				END_CASE
				%MW1300:=LEN(STR:= 转发转存);
			END_IF
			
			
			IF R_TRIG[6].Q THEN
				泵站位符:=FALSE;
				转发转存:='';
				%MW1300:=128;
				上液计数:=上液计数+1;
				IF 上液计数>=Expand_up_liquid_count THEN
					上液计数:=0;
					CASE Expand_Group OF
						1:
							CASE Expand_Number OF
								1:
									展缸1进液电池阀1自动:=FALSE;
									;
								2:
									展缸1进液电池阀2自动:=FALSE;
									
								3:
									展缸1进液电池阀3自动:=FALSE;
									
								4:
									展缸1进液电池阀4自动:=FALSE;
									
							END_CASE
						2:
							CASE Expand_Number OF
								1:
									展缸2进液电池阀1自动:=FALSE;
									
								2:
									展缸2进液电池阀2自动:=FALSE;
									
								3:
									展缸2进液电池阀3自动:=FALSE;
									
								4:
									展缸2进液电池阀4自动:=FALSE;
									
							END_CASE
						END_CASE
					Expand_up_liquid_OK:=TRUE; bActionDone:=TRUE;
					上液step:=0;
				ELSE
					上液step:=10;
				END_IF
			END_IF	
    END_CASE	
END_IF
END_ACTION

ACTION A10_init_初始化:
R_TRIG[1](CLK:=%MX2005.5 , Q=> );  //泵空闲中
R_TRIG[2](CLK:=%MX2005.5 , Q=> );  //泵空闲中

CASE 初始化step OF
	0:
		润洗展缸STEP:=0;
		清洗STEP:=0;
		上液step:=0;
		放硅胶板step:=0;
// 		展开step:=0;
		expand_initialization_OK:=FALSE;
		Expand_Group_clean_OK:=FALSE;
		Expand_up_liquid_OK:=FALSE;
		Expand_silica_gel_plate_OK:=FALSE;
		CASE Expand_Group OF
			1:
				CASE Expand_Number OF
					1:
						展缸1气缸1手动:=FALSE;
						展缸1气缸1自动:=FALSE;
						展缸1进液电池阀1手动:=FALSE;
						展缸1进液电池阀1自动:=FALSE;
						展缸1排液电池阀1手动:=FALSE;
						展缸1排液电池阀1自动:=FALSE;
						展缸1吹气电池阀1手动:=FALSE;
						展缸1吹气电池阀1自动:=FALSE;
					2:
						展缸1气缸2手动:=FALSE;
						展缸1气缸2自动:=FALSE;
						展缸1进液电池阀2手动:=FALSE;
						展缸1进液电池阀2自动:=FALSE;
						展缸1排液电池阀2手动:=FALSE;
						展缸1排液电池阀2自动:=FALSE;
						展缸1吹气电池阀2手动:=FALSE;
						展缸1吹气电池阀2自动:=FALSE;	
					3:
						展缸1气缸3手动:=FALSE;
						展缸1气缸3自动:=FALSE;
						展缸1进液电池阀3手动:=FALSE;
						展缸1进液电池阀3自动:=FALSE;	
						展缸1排液电池阀3手动:=FALSE;
						展缸1排液电池阀3自动:=FALSE;
						展缸1吹气电池阀3手动:=FALSE;
						展缸1吹气电池阀3自动:=FALSE;	
					4:
						展缸1气缸4手动:=FALSE;
						展缸1气缸4自动:=FALSE;
						展缸1进液电池阀4手动:=FALSE;
						展缸1进液电池阀4自动:=FALSE;	
						展缸1排液电池阀4手动:=FALSE;
						展缸1排液电池阀4自动:=FALSE;
						展缸1吹气电池阀4手动:=FALSE;
						展缸1吹气电池阀4自动:=FALSE;	
				END_CASE
				IF %MW1300=0 AND 泵站位符=FALSE  THEN
					转发转存:='/1Z0,2,2R$R';     //泵初始化指令 
					%MW1300:=LEN(STR:= 转发转存);   //发送字节数
					泵站位符:=TRUE;
					初始化STEP:=10;
				END_IF
			2:
				CASE Expand_Number OF
					1:
						展缸2气缸1手动:=FALSE;
						展缸2气缸1自动:=FALSE;
						展缸2进液电池阀1手动:=FALSE;
						展缸2进液电池阀1自动:=FALSE;
						展缸2排液电池阀1手动:=FALSE;
						展缸2排液电池阀1自动:=FALSE;
						展缸2吹气电池阀1手动:=FALSE;
						展缸2吹气电池阀1自动:=FALSE;
					2:
						展缸2气缸2手动:=FALSE;
						展缸2气缸2自动:=FALSE;
						展缸2进液电池阀2手动:=FALSE;
						展缸2进液电池阀2自动:=FALSE;
						展缸2排液电池阀2手动:=FALSE;
						展缸2排液电池阀2自动:=FALSE;
						展缸2吹气电池阀2手动:=FALSE;
						展缸2吹气电池阀2自动:=FALSE;	
					3:
						展缸2气缸3手动:=FALSE;
						展缸2气缸3自动:=FALSE;
						展缸2进液电池阀3手动:=FALSE;
						展缸2进液电池阀3自动:=FALSE;	
						展缸2排液电池阀3手动:=FALSE;
						展缸2排液电池阀3自动:=FALSE;
						展缸2吹气电池阀3手动:=FALSE;
						展缸2吹气电池阀3自动:=FALSE;	
					4:
						展缸2气缸4手动:=FALSE;
						展缸2气缸4自动:=FALSE;
						展缸2进液电池阀4手动:=FALSE;
						展缸2进液电池阀4自动:=FALSE;	
						展缸2排液电池阀4手动:=FALSE;
						展缸2排液电池阀4自动:=FALSE;
						展缸2吹气电池阀4手动:=FALSE;
						展缸2吹气电池阀4自动:=FALSE;
				END_CASE 
				 IF %MW1300=0 AND 泵站位符=FALSE  THEN
					转发转存:='/2Z0,2,2R$R';     //泵初始化指令 
					%MW1300:=LEN(STR:= 转发转存);   //发送字节数
					泵站位符:=TRUE;
					初始化STEP:=10;
				END_IF
		END_CASE

	
		
		
	10:
		CASE Expand_Group OF
			1:
				IF %MW1300=0 THEN
					转发转存:='/1Q$R';          //查询泵状态指令
					%MW1300:=LEN(STR:= 转发转存);
				END_IF
				
				
				IF R_TRIG[1].Q THEN
					泵初始化完成:=TRUE;
					泵站位符:=FALSE;
					初始化STEP:=0; bActionDone:=TRUE;
				END_IF
			2:
				IF %MW1300=0 THEN
					转发转存:='/2Q$R';          //查询泵状态指令
					%MW1300:=LEN(STR:= 转发转存);
				END_IF
				
				IF R_TRIG[2].Q THEN
					泵初始化完成:=TRUE;
					泵站位符:=FALSE;
					初始化STEP:=0; bActionDone:=TRUE;
				END_IF
		END_CASE
END_CASE
END_ACTION

ACTION A26_rinse_suction:
(* 润洗展缸-抽吸: 真空由上位机 Pump_L2 提供 (本动作前置 vacuum_on).
   等废液抽净 -> 关进液阀/开吹气阀 -> 吹气定时 -> 关阀完成. 阀状态承接 A21_rinse 注液. *)
TON[10](IN:=(Expand_Group=1 AND  展缸1溶剂废液检测传感器) OR (Expand_Group=2 AND  展缸2溶剂废液检测传感器),PT:=T#10S);
TON_2(IN:=润洗展缸STEP=0, PT:=T#3S);
TON[4](IN:=润洗展缸STEP=10,PT:=T#30S);
TON[7](IN:=润洗展缸STEP=0, PT:=T#60S);   (* 抽吸超时看门狗 *)
CASE 润洗展缸STEP OF
	0:
		IF TON_2.Q THEN
			IF TON[10].Q THEN
				CASE Expand_Group OF
					1:
						CASE Expand_Number OF
							1:
								展缸1进液电池阀1自动:=FALSE;
								展缸1吹气电池阀1自动:=TRUE;
								润洗展缸STEP:=10;
							2:
								展缸1进液电池阀2自动:=FALSE;
								展缸1吹气电池阀2自动:=TRUE;
								润洗展缸STEP:=10;
							3:
								展缸1进液电池阀3自动:=FALSE;
								展缸1吹气电池阀3自动:=TRUE;
								润洗展缸STEP:=10;
							4:
								展缸1进液电池阀4自动:=FALSE;
								展缸1吹气电池阀4自动:=TRUE;
								润洗展缸STEP:=10;
						END_CASE
					2:
						CASE Expand_Number OF
							1:
								展缸2进液电池阀1自动:=FALSE;
								展缸2吹气电池阀1自动:=TRUE;
								润洗展缸STEP:=10;
							2:
								展缸2进液电池阀2自动:=FALSE;
								展缸2吹气电池阀2自动:=TRUE;
								润洗展缸STEP:=10;
							3:
								展缸2进液电池阀3自动:=FALSE;
								展缸2吹气电池阀3自动:=TRUE;
								润洗展缸STEP:=10;
							4:
								展缸2进液电池阀4自动:=FALSE;
								展缸2吹气电池阀4自动:=TRUE;
								润洗展缸STEP:=10;
						END_CASE
				END_CASE
			ELSIF TON[7].Q THEN
				Develop_L2_ErrorCode:=402;   (* 抽吸超时: 废液未抽净 *)
				润洗展缸STEP:=0;
				bActionError:=TRUE;
			END_IF
		END_IF
	10:
		IF TON[4].Q THEN
			CASE Expand_Group OF
				1:
					CASE Expand_Number OF
					1:
						展缸1排液电池阀1自动:=FALSE;
						展缸1吹气电池阀1自动:=FALSE;
						Expand_Group_clean_OK:=TRUE; bActionDone:=TRUE;
						润洗展缸STEP:=0;
					2:
						展缸1排液电池阀2自动:=FALSE;
						展缸1吹气电池阀2自动:=FALSE;
						Expand_Group_clean_OK:=TRUE; bActionDone:=TRUE;
						润洗展缸STEP:=0;
					3:
						展缸1排液电池阀3自动:=FALSE;
						展缸1吹气电池阀3自动:=FALSE;
						Expand_Group_clean_OK:=TRUE; bActionDone:=TRUE;
						润洗展缸STEP:=0;
					4:
						展缸1排液电池阀4自动:=FALSE;
						展缸1吹气电池阀4自动:=FALSE;
						Expand_Group_clean_OK:=TRUE; bActionDone:=TRUE;
						润洗展缸STEP:=0;
					END_CASE
				2:
					CASE Expand_Number OF
					1:
						展缸2排液电池阀1自动:=FALSE;
						展缸2吹气电池阀1自动:=FALSE;
						Expand_Group_clean_OK:=TRUE; bActionDone:=TRUE;
						润洗展缸STEP:=0;
					2:
						展缸2排液电池阀2自动:=FALSE;
						展缸2吹气电池阀2自动:=FALSE;
						Expand_Group_clean_OK:=TRUE; bActionDone:=TRUE;
						润洗展缸STEP:=0;
					3:
						展缸2排液电池阀3自动:=FALSE;
						展缸2吹气电池阀3自动:=FALSE;
						Expand_Group_clean_OK:=TRUE; bActionDone:=TRUE;
						润洗展缸STEP:=0;
					4:
						展缸2排液电池阀4自动:=FALSE;
						展缸2吹气电池阀4自动:=FALSE;
						Expand_Group_clean_OK:=TRUE; bActionDone:=TRUE;
						润洗展缸STEP:=0;
					END_CASE
			END_CASE
		END_IF
END_CASE
END_ACTION

END_PROGRAM

// Device/Application/50_action/PhotoScrape_L2
PROGRAM PhotoScrape_L2
VAR
	初始化step: INT;
	拍照step: INT;
	刮板收集step: INT;
	bActionDone: BOOL;
	bActionError: BOOL;
	L2_StartTrig: R_TRIG;
END_VAR

(* PhotoScrape 工位 L2 统一动作派发器
   按 PhotoScrape_L2_ActionCode 派发到纯设备原子动作 (不含机器人/相机/CNC 握手).
   Start 上升沿接受请求 -> RUNNING 每周期调用对应原子 -> bActionDone=DONE / bActionError=ERROR. *)
L2_StartTrig(CLK := PhotoScrape_L2_Start);

CASE PhotoScrape_L2_State OF
	0:  (* IDLE *)
		PhotoScrape_L2_Step := 0;
		IF L2_StartTrig.Q THEN
			PhotoScrape_L2_AcceptedSeq := PhotoScrape_L2_RequestSeq;
			PhotoScrape_L2_ActiveCode  := PhotoScrape_L2_ActionCode;
			PhotoScrape_L2_ErrorCode   := 0;
			PhotoScrape_L2_Retryable   := FALSE;
			bActionDone  := FALSE;
			bActionError := FALSE;
			初始化step := 0;
			拍照step := 0;
			刮板收集step := 0;
			CASE PhotoScrape_L2_ActionCode OF
				10, 31, 32, 33, 34, 35, 36, 40, 41, 51, 52:
					PhotoScrape_L2_SafeState := 0;
					PhotoScrape_L2_State     := 10;   (* RUNNING *)
			ELSE
				PhotoScrape_L2_ErrorCode    := 101;  (* 未知动作码 *)
				PhotoScrape_L2_Retryable    := TRUE;
				PhotoScrape_L2_CompletedSeq := PhotoScrape_L2_AcceptedSeq;
				PhotoScrape_L2_State        := 30;   (* REJECTED *)
			END_CASE
		END_IF

	10: (* RUNNING *)
		IF PhotoScrape_L2_Reset THEN PhotoScrape_L2_State := 0; RETURN; END_IF   (* RUNNING 中 RESET: 中止挂死动作 *)
		CASE PhotoScrape_L2_ActiveCode OF
			10: A10_init_初始化();
			31: A31_cam_移轴335();
			32: A32_cam_定位();
			33: A33_cam_下压();
			36: 粉末收集器定位自动:=PhotoScrape_PowderCollectorLocate_Target; bActionDone:=TRUE;
			34: A34_cam_相机位();
			35: A35_cam_回零();
			40: A40_scrape_刮取();
			41: A41_scrape_收尾();
			51: A51_取料松压();
			52: A52_取料停旋转();
		END_CASE
		IF bActionDone THEN
			bActionDone              := FALSE;
			PhotoScrape_L2_CompletedSeq := PhotoScrape_L2_AcceptedSeq;
			PhotoScrape_L2_State        := 20;   (* DONE *)
		ELSIF bActionError THEN              (* 设备预条件未满足 -> 报错交上位机 *)
			bActionError             := FALSE;
			PhotoScrape_L2_Retryable    := TRUE;
			PhotoScrape_L2_CompletedSeq := PhotoScrape_L2_AcceptedSeq;
			PhotoScrape_L2_State        := 40;   (* ERROR; ErrorCode 由原子置 *)
		END_IF

	20, 30, 40, 50:  (* 终态: 等 Start 落沿或 Reset 回 IDLE *)
		IF (NOT PhotoScrape_L2_Start) OR PhotoScrape_L2_Reset THEN
			PhotoScrape_L2_State := 0;
		END_IF
END_CASE

ACTION A10_init_初始化:





CASE 初始化step OF
	0:
		刮板拍照真空自动:=FALSE;
		刮板拍照真空手动:=FALSE;
		刮板拍照无刷电机手动:=FALSE;
		刮板拍照无刷电机自动:=FALSE;
		刮板拍照定位气缸手动:=FALSE;
		刮板拍照定位气缸自动:=FALSE;
		粉末收集器定位手动:=FALSE;
		粉末收集器定位自动:=FALSE;
		刮板拍照遮光气缸手动:=FALSE;
		刮板拍照遮光气缸自动:=FALSE;
		刮板拍照旋转气缸手动:=FALSE;
		刮板拍照旋转气缸自动:=FALSE;
		刮板拍照下压气缸手动:=FALSE;
		刮板拍照下压气缸自动:=FALSE;
		
		
	
		
		拍照step:=0;
// 		机器人取物料step:=0;
		刮板收集step:=0;
		
		Camera_scraper_initialization_OK:=FALSE;
		Photo_preparation_completed_OK:=FALSE;
		Scraper_collection_completed:=FALSE;
		Robot_completes_material_retrieval:=FALSE;
		初始化step:=5;
	5:
		刮板轴10ZDATE.xMoveAbs:=FALSE;
		刮板轴9XDATE.xMoveAbs:=FALSE;
		拍照轴8YDATE.xMoveAbs:=FALSE;
		初始化step:=6;
	6:
		刮板轴10ZDATE.fAbsTarget:=0;
		刮板轴10ZDATE.xMoveAbs:=TRUE;
		IF 刮板轴10ZDATE.bAbMoveDone THEN
			刮板轴10ZDATE.xMoveAbs:=FALSE;
			初始化step:=10;
		END_IF
	10:
		刮板轴9XDATE.fAbsTarget:=335;
		刮板轴9XDATE.xMoveAbs:=TRUE;
		IF 刮板轴9XDATE.bAbMoveDone THEN
			刮板轴9XDATE.xMoveAbs:=FALSE;
			初始化step:=20;
		END_IF
	20:
		IF 刮板拍照遮光气缸上位 THEN
			拍照轴8YDATE.fAbsTarget:=0;
			拍照轴8YDATE.xMoveAbs:=TRUE;
			IF 拍照轴8YDATE.bAbMoveDone THEN
				拍照轴8YDATE.xMoveAbs:=FALSE;
				Camera_scraper_initialization_OK:=TRUE; bActionDone:=TRUE;
				初始化step:=0;
			END_IF	
		END_IF		
	
END_CASE
END_ACTION

ACTION A32_cam_定位:
(* 拍照定位气缸夹紧 (上位机已驱动机器人放板) *)
刮板拍照定位气缸自动:=PhotoScrape_CamLocate_Target;
bActionDone:=TRUE;
END_ACTION

ACTION A35_cam_回零:
(* 遮光上 + 拍照Y轴回零 (上位机已拍照完成) *)
CASE 拍照step OF
	0:
		刮板拍照遮光气缸自动:=FALSE;
		拍照step:=10;
	10:
		IF 刮板拍照遮光气缸上位 THEN
			拍照轴8YDATE.fAbsTarget:=0;
			拍照轴8YDATE.xMoveAbs:=TRUE;
			拍照step:=20;
		END_IF
	20:
		IF 拍照轴8YDATE.bAbMoveDone THEN
			拍照轴8YDATE.xMoveAbs:=FALSE;
			拍照step:=0;
			bActionDone:=TRUE;
		END_IF
END_CASE
END_ACTION

ACTION A34_cam_相机位:
(* 移到相机位 + 遮光下 (随后由上位机视觉控制器拍照) *)
CASE 拍照step OF
	0:
		IF 刮板拍照遮光气缸上位 THEN
// 			拍照轴8YDATE.fAbsTarget:=420;
			拍照轴8YDATE.fAbsTarget:=Photo_8Y_Target;
			拍照轴8YDATE.xMoveAbs:=TRUE;
			拍照step:=10;
		END_IF
	10:
		IF 拍照轴8YDATE.bAbMoveDone THEN
			拍照轴8YDATE.xMoveAbs:=FALSE;
			刮板拍照遮光气缸自动:=TRUE;
			拍照step:=20;
		END_IF
	20:
		IF 刮板拍照遮光气缸下位 THEN
			拍照step:=0;
			bActionDone:=TRUE;
		END_IF
END_CASE
END_ACTION

ACTION A33_cam_下压:
(* PhotoScrape press cylinder target: TRUE=press down, FALSE=release/up *)
IF PhotoScrape_CamPress_Target THEN
	刮板拍照下压气缸自动:=TRUE;
	bActionDone:=TRUE;
ELSE
	刮板拍照下压气缸自动:=FALSE;
	IF 刮板拍照下压气缸上位 THEN
		bActionDone:=TRUE;
	END_IF
END_IF
END_ACTION

ACTION A31_cam_移轴335:
(* 刮板X轴到放板/上料位 335 *)
刮板轴9XDATE.fAbsTarget:=335;
刮板轴9XDATE.xMoveAbs:=TRUE;
IF 刮板轴9XDATE.bAbMoveDone THEN
	刮板轴9XDATE.xMoveAbs:=FALSE;
	bActionDone:=TRUE;
END_IF
END_ACTION

ACTION A40_scrape_刮取:
(* 刮取单 pass: 上位机已写 g_pass_z 等 g_* 参数; 触发 PLC_CNC 跑一刀
   CNC启动/CNC完成 为 PLC 内部 SoftMotion 触发线 (保留); 多 pass 由上位机循环调用本动作 *)
CASE 刮板收集step OF
	0:
		刮板拍照真空自动:=TRUE;
		CNC启动:=TRUE;
		刮板收集step:=10;
	10:
		IF CNC完成 THEN
			CNC启动:=FALSE;
			刮板收集step:=0;
			bActionDone:=TRUE;
		END_IF
END_CASE
END_ACTION

ACTION A52_取料停旋转:
(* 取料收尾: 停旋转气缸 (上位机已驱动机器人退出取走收集器) *)
刮板拍照旋转气缸自动:=FALSE;
bActionDone:=TRUE;
END_ACTION

ACTION A51_取料松压:
(* 取料: 松下压气缸 (上位机已驱动机器人到收集器夹持位) *)
刮板拍照下压气缸自动:=FALSE;
IF 刮板拍照下压气缸上位 THEN
	bActionDone:=TRUE;
END_IF
END_ACTION

ACTION A41_scrape_收尾:
(* 刮取收尾: 关真空/电机, 旋转气缸翻转倒料; 定位释放由 locate_cylinder(FALSE) 统一处理 *)
刮板拍照真空自动:=FALSE;
刮板拍照无刷电机自动:=FALSE;
刮板拍照旋转气缸自动:=TRUE;
bActionDone:=TRUE;
END_ACTION

END_PROGRAM

// Device/Application/30_Ethercat任务/PLC_CNC
PROGRAM PLC_CNC
VAR
	SMC_Interpolator: SMC_Interpolator;
	SMC_ControlAxisByPos1: SMC_ControlAxisByPos;
	SMC_ControlAxisByPos2: SMC_ControlAxisByPos;
	SMC_ControlAxisByPos3: SMC_ControlAxisByPos;
	SMC_TRAFO_Gantry3: SMC_TRAFO_Gantry3;
	SMC_TRAFOF_Gantry3: SMC_TRAFOF_Gantry3;
	SMC_NCDecoder_0: SMC_NCDecoder;
	SMC_CheckVelocities: SMC_CheckVelocities;
	SMC_SmoothPath: SMC_SmoothPath;
	SR: SR;
	RS: RS;
END_VAR
VAR // added by the converter: edge detectors and wires of the graphical bodies
    _w1, _w2, _w3 : BOOL;
    _w4, _w5 : ANY;
END_VAR

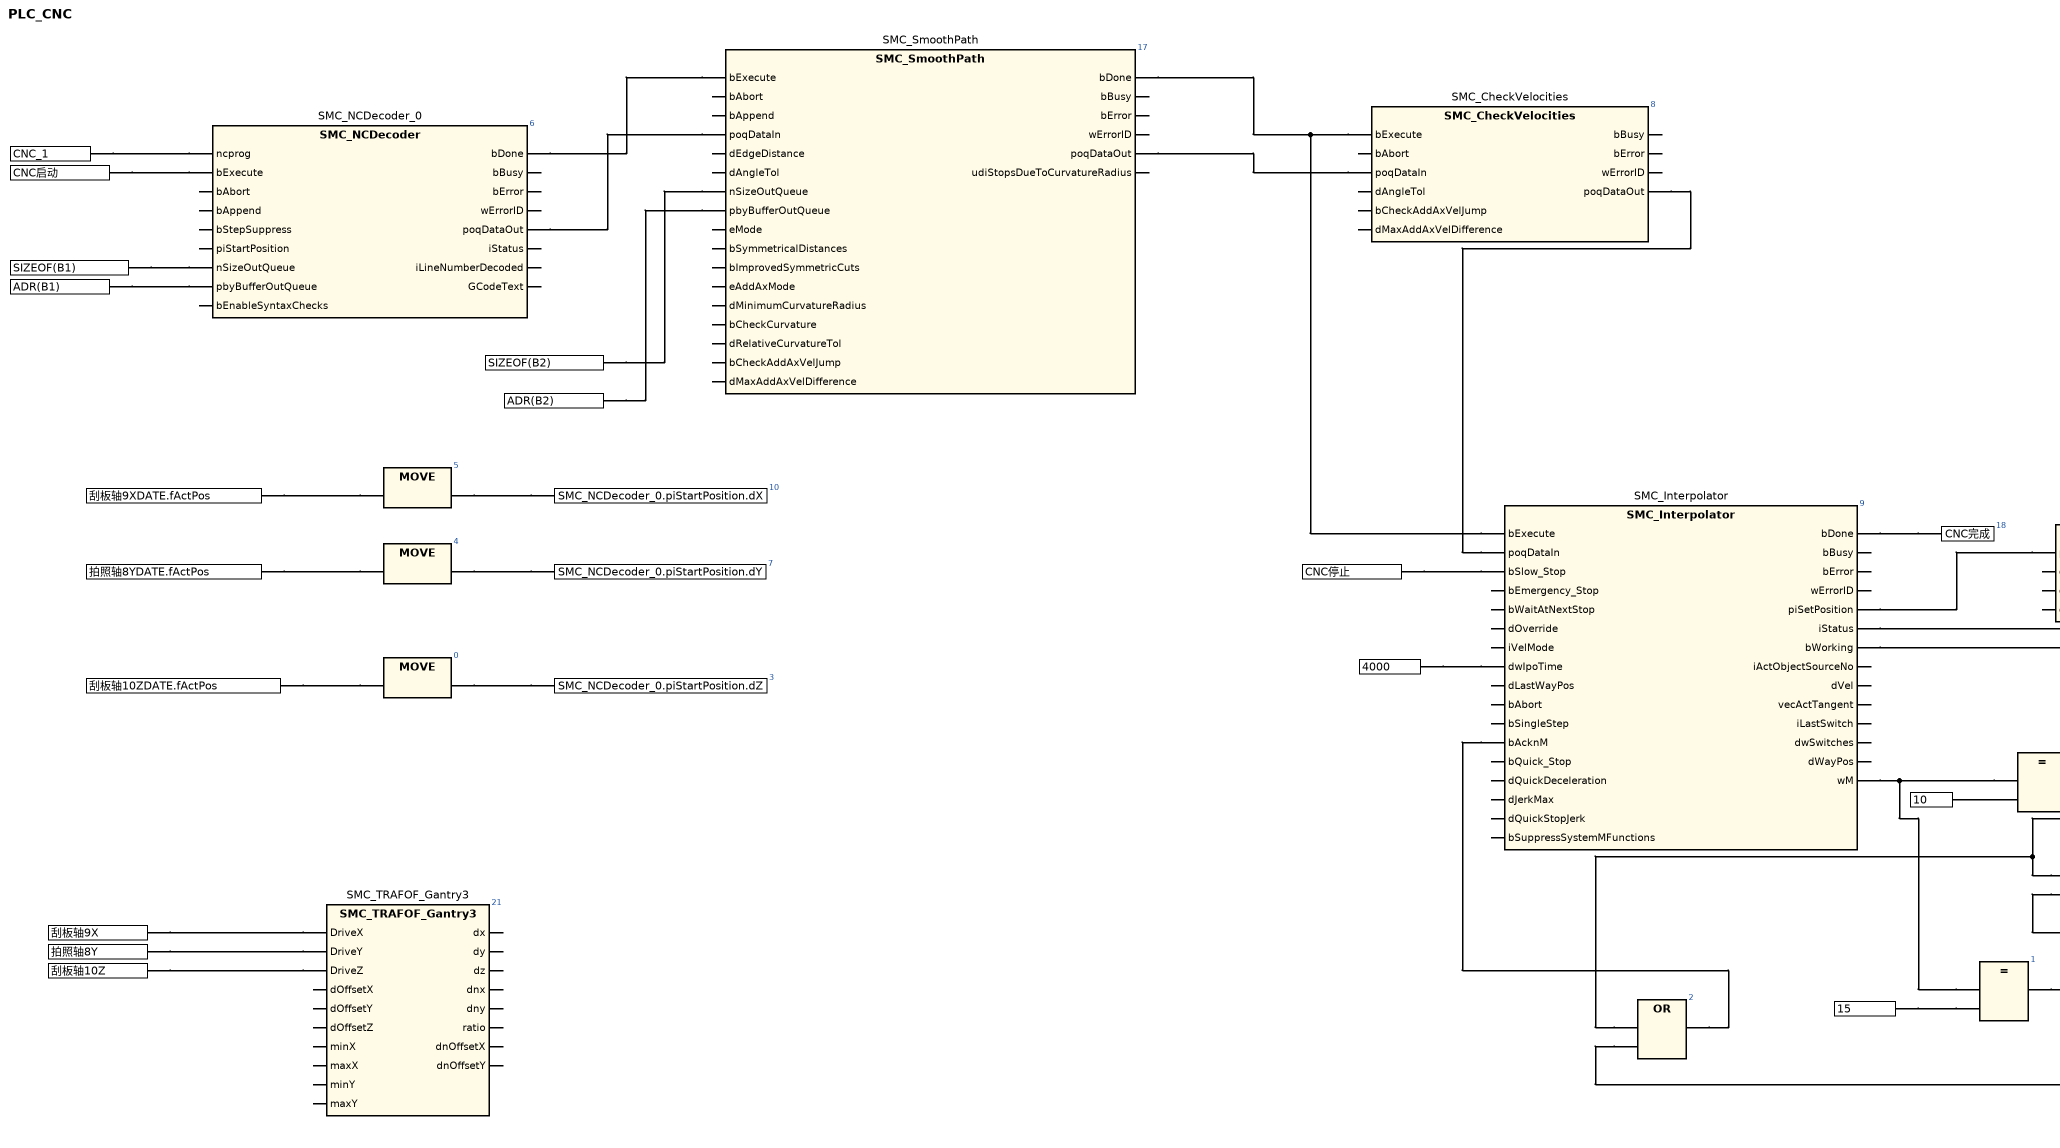
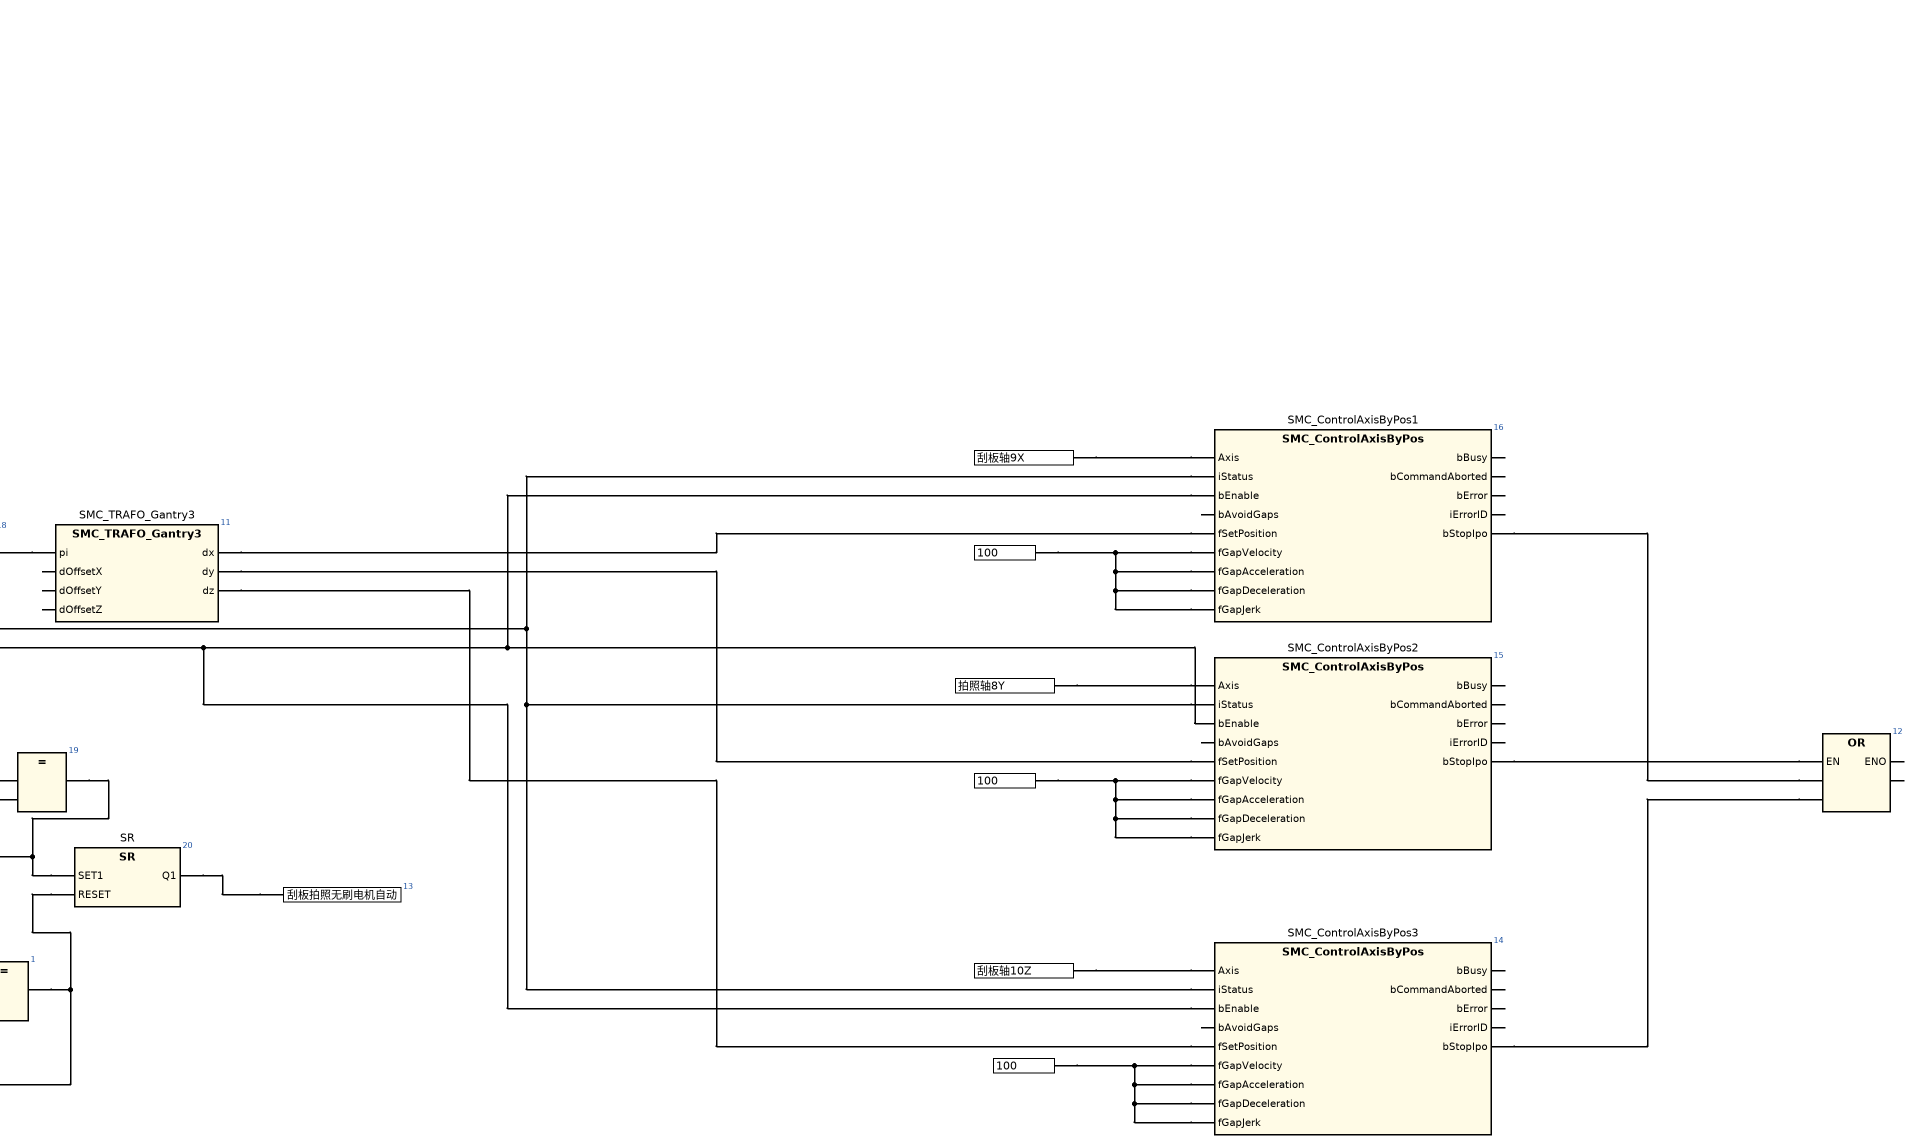
// note: 4 stored wires end on pins the file does not list and are not shown
_w1 := SMC_Interpolator.wM = 15;
_w3 := _w2 OR _w1;
SMC_NCDecoder_0.piStartPosition.dZ := 刮板轴10ZDATE.fActPos;
_w4 := 拍照轴8YDATE.fActPos;
_w5 := 刮板轴9XDATE.fActPos;
SMC_NCDecoder_0(
    ncprog := CNC_1,
    bExecute := CNC启动,
    nSizeOutQueue := SIZEOF(B1),
    pbyBufferOutQueue := ADR(B1)); // SMC_NCDecoder
SMC_NCDecoder_0.piStartPosition.dY := _w4;
SMC_CheckVelocities(bExecute := SMC_SmoothPath.bDone, poqDataIn := SMC_SmoothPath.poqDataOut);
SMC_Interpolator(
    bExecute := SMC_SmoothPath.bDone,
    poqDataIn := SMC_CheckVelocities.poqDataOut,
    bSlow_Stop := CNC停止,
    dwIpoTime := 4000,
    bAcknM := _w3);
SMC_NCDecoder_0.piStartPosition.dX := _w5;
SMC_TRAFO_Gantry3(pi := SMC_Interpolator.piSetPosition);
IF SMC_ControlAxisByPos2.bStopIpo THEN (* SMC_ControlAxisByPos1.bStopIpo OR SMC_ControlAxisByPos3.bStopIpo; result not used *) END_IF
刮板拍照无刷电机自动 := SR.Q1;
SMC_ControlAxisByPos3(
    Axis := 刮板轴10Z,
    iStatus := SMC_Interpolator.iStatus,
    bEnable := SMC_Interpolator.bWorking,
    fSetPosition := SMC_TRAFO_Gantry3.dz,
    fGapVelocity := 100,
    fGapAcceleration := 100,
    fGapDeceleration := 100,
    fGapJerk := 100); // SMC_ControlAxisByPos
SMC_ControlAxisByPos2(
    Axis := 拍照轴8Y,
    iStatus := SMC_Interpolator.iStatus,
    bEnable := SMC_Interpolator.bWorking,
    fSetPosition := SMC_TRAFO_Gantry3.dy,
    fGapVelocity := 100,
    fGapAcceleration := 100,
    fGapDeceleration := 100,
    fGapJerk := 100); // SMC_ControlAxisByPos
SMC_ControlAxisByPos1(
    Axis := 刮板轴9X,
    iStatus := SMC_Interpolator.iStatus,
    bEnable := SMC_Interpolator.bWorking,
    fSetPosition := SMC_TRAFO_Gantry3.dx,
    fGapVelocity := 100,
    fGapAcceleration := 100,
    fGapDeceleration := 100,
    fGapJerk := 100); // SMC_ControlAxisByPos
SMC_SmoothPath(
    bExecute := SMC_NCDecoder_0.bDone,
    poqDataIn := SMC_NCDecoder_0.poqDataOut,
    nSizeOutQueue := SIZEOF(B2),
    pbyBufferOutQueue := ADR(B2));
CNC完成 := SMC_Interpolator.bDone;
_w2 := SMC_Interpolator.wM = 10;
SR(SET1 := _w2, RESET := _w1);
SMC_TRAFOF_Gantry3(DriveX := 刮板轴9X, DriveY := 拍照轴8Y, DriveZ := 刮板轴10Z);

END_PROGRAM

// Device/Application/25_FB_功能块/FB_Mode
FUNCTION_BLOCK FB_Mode
VAR_INPUT
    xStart      : BOOL;  // 启动按钮
    xStop       : BOOL;  // 停止按钮
    xReset      : BOOL;  // 复位按钮
    xAutoMode   : BOOL;  // TRUE=自动模式，FALSE=手动模式
    xFault      : BOOL;  // 故障信号
    xEmergency  : BOOL;  // 急停信号（急停按下为FALSE）
END_VAR
VAR_OUTPUT
    bRed        : BOOL;  // 红灯
    bYellow     : BOOL;  // 黄灯
    bGreen      : BOOL;  // 绿灯
    bBuzzer     : BOOL;  // 蜂鸣器
    iState      : INT;   // 设备状态: 0=停止, 1=运行, 2=故障, 3=急停
    bAuto       : BOOL;  // 自动模式指示
END_VAR
VAR
    iDeviceState : INT := 0;  // 0=停止, 1=运行, 2=故障, 3=急停
    
    // 定时器
    tBuzzerPulse : TON;  // 蜂鸣器脉冲
    tFlashTimer  : TON;  // 闪烁定时器
    tShortBeep   : TON;  // 短鸣定时器
    tEmergencyBeep : TON; // 急停蜂鸣器定时器
	// 蜂鸣器激活
	tEmergencyBeep1: TON;
    
    // 标志
    bBuzzerActive : BOOL := FALSE;  // 蜂鸣器激活
    bFlashFlag    : BOOL;           // 闪烁标志
    bBeepOnce     : BOOL := FALSE;  // 单次蜂鸣标志
    bEmergencyBuzzer : BOOL := FALSE; // 急停蜂鸣器标志
    bEmergencyActive : BOOL := FALSE; // 急停激活标志
	ALT_0: ALT;
	ALT_1: ALT;
	TON_0: TON;
	ALT_2: ALT;
	TON_1: TON;
	TON_2: TON;
END_VAR
VAR_INPUT
	bWarning_alarm: BOOL;
END_VAR

// 模式状态
bAuto := xAutoMode;

// 状态机
CASE iDeviceState OF
    EN_功能块状态.停止:  // 停止状态
        IF NOT xEmergency THEN
            iDeviceState := EN_功能块状态.急停;  // 急停
            bEmergencyActive := TRUE;
        ELSIF xFault THEN
            iDeviceState := EN_功能块状态.故障;  // 故障
            bBuzzerActive := TRUE;
        ELSIF (bAuto AND xStart)  THEN
		 bBeepOnce := TRUE;  // 启动短鸣
		  iDeviceState := EN_功能块状态.初始化;  // 初始化

        END_IF;
    
    EN_功能块状态.运行:  // 运行状态
        IF NOT xEmergency THEN
            iDeviceState := EN_功能块状态.急停;  // 急停
            bEmergencyActive := TRUE;
        ELSIF xFault THEN
            iDeviceState := EN_功能块状态.故障;  // 故障
            bBuzzerActive := TRUE;
        ELSIF xStop THEN
            iDeviceState := EN_功能块状态.停止;  // 停止
            bBeepOnce := TRUE;  // 停止短鸣
        END_IF;
        
    EN_功能块状态.故障:  // 故障状态
        IF NOT xEmergency THEN
            iDeviceState := EN_功能块状态.急停;  // 急停
            bEmergencyActive := TRUE;
        ELSIF xReset AND NOT xFault THEN
            iDeviceState := EN_功能块状态.停止;  // 停止
            bBuzzerActive := FALSE;
			bBuzzer:=FALSE;
        END_IF;
        
    EN_功能块状态.急停:  // 急停状态
        // 急停复位需要：急停信号解除 + 复位按钮按下
        IF  xEmergency AND xReset THEN
            iDeviceState := EN_功能块状态.停止;  // 停止
            bEmergencyActive := FALSE;
            bEmergencyBuzzer := FALSE;
			bBuzzer:=FALSE;
        END_IF;
	EN_功能块状态.初始化:  //初始化状态
	 TON_0(IN:=TRUE , PT:=T#3S );
		IF TON_0.Q THEN
		iDeviceState := EN_功能块状态.运行;  // 运行
		END_IF 
END_CASE;

// 急停蜂鸣器控制（急停时蜂鸣器以不同频率鸣响）
IF  bEmergencyActive THEN
    tEmergencyBeep(IN := NOT tEmergencyBeep.Q, PT := T#2S );
	ALT_1(xExecute:= tEmergencyBeep.Q, xOut:=bBuzzer );  // 急停时蜂鸣器响2秒，停2秒	
END_IF;

//三色灯控制
// 闪烁定时器
tFlashTimer(IN := NOT tFlashTimer.Q, PT := T#500MS);
ALT_0(xExecute:=tFlashTimer.Q , xOut:=bFlashFlag );

CASE iDeviceState OF
    EN_功能块状态.停止:  // 停止状态
        IF bAuto THEN
            bYellow := TRUE;           // 自动模式：黄灯常亮
        ELSE
            bYellow := bFlashFlag;     // 手动模式：黄灯闪烁
        END_IF;
		 bGreen :=FALSE;
		 bRed :=FALSE;
        
    EN_功能块状态.运行:  // 运行状态
        bGreen := TRUE;
         bRed :=FALSE;
		  bYellow := FALSE; 
    EN_功能块状态.故障:  // 故障状态
        bRed := TRUE;
         bGreen :=FALSE;
		 bYellow := FALSE; 
    EN_功能块状态.急停:  // 急停状态
        bRed := bFlashFlag;  // 红灯闪烁
		bGreen :=FALSE;
		 bYellow := FALSE; 
END_CASE;
tShortBeep(IN := bBeepOnce AND NOT bEmergencyActive, PT := T#500MS);
// 蜂鸣器控制
IF bBeepOnce AND NOT bEmergencyActive THEN
	bBuzzer := TRUE;  // 短鸣
    IF tShortBeep.Q THEN
        bBeepOnce := FALSE;
       bBuzzer := FALSE;
    END_IF;
    
END_IF;

// 故障时蜂鸣器（非急停状态时生效）
IF NOT bEmergencyActive AND xFault  THEN
    tBuzzerPulse(IN := NOT tBuzzerPulse.Q, PT := T#500MS);
ALT_2(xExecute:= tBuzzerPulse.Q, xOut:= bBuzzer);
END_IF;


//蜂鸣器5S后停止
TON_2(IN:=iDeviceState=2 OR iDeviceState=3 OR bWarning_alarm ,PT:=T#5S);
IF TON_2.Q THEN
	bBuzzer:=FALSE;
END_IF

IF bWarning_alarm AND NOT TON_2.Q THEN
	bBuzzer:=TRUE;
	
END_IF
IF bWarning_alarm  THEN
	 bRed := TRUE;
	  
END_IF

IF xReset THEN
	bBuzzer:=FALSE;
	bRed := FALSE;
END_IF



// 输出状态
iState := iDeviceState;

END_FUNCTION_BLOCK

// Device/Application/30_Ethercat任务/PLC_Servo_伺服
PROGRAM PLC_Servo_伺服
VAR
	FB_SERVOAXIS_0: FB_SERVOAXIS;
	FB_SERVOAXIS_1: FB_SERVOAXIS;
	FB_SERVOAXIS_2: FB_SERVOAXIS;
	FB_SERVOAXIS_3: FB_SERVOAXIS;
	FB_SERVOAXIS_4: FB_SERVOAXIS;
	FB_SERVOAXIS_5: FB_SERVOAXIS;
	FB_SERVOAXIS_6: FB_SERVOAXIS;
	FB_SERVOAXIS_7: FB_SERVOAXIS;
	FB_SERVOAXIS_8: FB_SERVOAXIS;
	FB_SERVOAXIS_9: FB_SERVOAXIS;
	FB_SERVOAXIS_10: FB_SERVOAXIS;
	HOME_1STEP: INT;
	HOME_2STEP: INT;
	i: INT;
	FB_Teach_1: FB_Teach;
	FB_Teach_2: FB_Teach;
	FB_Teach_3: FB_Teach;
	FB_Teach_4: FB_Teach;
	FB_Teach_5: FB_Teach;
	FB_Teach_6: FB_Teach;
	n: INT;
	TON_SysReset: TON;
	bSysResetDone: BOOL;
	TON_CyInhibit: TON;
	bCyInhibitDone: BOOL;
	TON_AutoHome: TON;
	bAutoHomeDone: BOOL;
	TON_AutoHomeReset: TON;
	bAutoHomeReq: BOOL;
	bAutoHomeOnly45: BOOL;
	bAllHomed: BOOL;
	R_TRIG_HomeAll: R_TRIG;
	R_TRIG_Home45: R_TRIG;
END_VAR

TON_SysReset(IN:= ethercat1.m_master.m_uiactualnoslaves=13 AND NOT bSysResetDone, PT:= T#3S);
bSysReset := (ethercat1.m_master.m_uiactualnoslaves=13) AND NOT bSysResetDone;
IF TON_SysReset.Q THEN
	bSysResetDone := TRUE;
END_IF

//开机气缸超时抑制窗(等气压/传感器稳定, 一次性, 上电/下载重新触发); 消费在 PLC_MainPRG 清 cyinderAlarm
TON_CyInhibit(IN:= ethercat1.m_master.m_uiactualnoslaves=13 AND NOT bCyInhibitDone, PT:= T#15S);
bCyInhibit := (ethercat1.m_master.m_uiactualnoslaves=13) AND NOT bCyInhibitDone;
IF TON_CyInhibit.Q THEN
	bCyInhibitDone := TRUE;
END_IF

//开机一次性自动回零触发(仅4X/5Z): 13从站OP + 急停释放 + 复位窗结束 + 上样两轴已使能, 延时确保驱动上电
TON_AutoHome(IN:= ethercat1.m_master.m_uiactualnoslaves=13 AND 急停 AND bSysResetDone
	AND 上样轴5Z轴DATE.bEnabled AND 上样轴4X轴DATE.bEnabled
	AND MODE_State<>1 AND NOT bAutoHomeDone, PT:= T#2S);
IF TON_AutoHome.Q AND NOT bAutoHomeDone THEN
	bAutoHomeReq := TRUE;
	bAutoHomeDone := TRUE;
END_IF

//开机自动回零完成 -> 拉1.5s复位窗, 设备从故障自动回到停止; 失败保持故障可见(不掩盖)
bAllHomed := 玻璃上料轴1ZDATE.bHomed AND 玻璃上料轴2ZDATE.bHomed AND 打样瓶上料轴3YDATE.bHomed
	AND 点样轴6XDATE.bHomed AND 点样轴7YDATE.bHomed AND 拍照轴8YDATE.bHomed
	AND 刮板轴9XDATE.bHomed AND 刮板轴10ZDATE.bHomed AND 地轨轴11YDATE.bHomed
	AND 上样轴4X轴DATE.bHomed AND 上样轴5Z轴DATE.bHomed;
IF bAutoHomeReq AND bAllHomed THEN
	TON_AutoHomeReset(IN:= TRUE, PT:= T#1500MS);
	bAutoHomeResetPulse := TRUE;
	IF TON_AutoHomeReset.Q THEN
		bAutoHomeReq := FALSE;
		bAutoHomeResetPulse := FALSE;
	END_IF
ELSE
	TON_AutoHomeReset(IN:= FALSE, PT:= T#1500MS);
	bAutoHomeResetPulse := FALSE;
END_IF

伺服调用 ();
//检测ECAT通讯连接数量
IF ethercat1.m_master.m_uiactualnoslaves<>13 THEN
	ECAT掉站报警:=TRUE;
	ELSE
	ECAT掉站报警:=FALSE;
END_IF

IF MODE_State<>1 THEN
	伺服一键回原点 ();
	IF NOT 点样测试 THEN
		位置示教 ();
	END_IF
	
END_IF

IF MODE_State=1 THEN		
	FOR n:=1 TO 10 BY 1 DO
		HMI_打样瓶上料轴3Y.execute[n]:=FALSE;
		HMI_打样瓶上料轴3Y.write[n]:=FALSE;
		HMI_点样轴6X.execute[n]:=FALSE;
		HMI_点样轴6X.write[n]:=FALSE;
		HMI_点样轴7Y.execute[n]:=FALSE;
		HMI_点样轴7Y.write[n]:=FALSE;
		HMI_地轨轴11Y.execute[n]:=FALSE;
		HMI_地轨轴11Y.write[n]:=FALSE;
		HMI_上样轴4X轴.execute[n]:=FALSE;
		HMI_上样轴4X轴.write[n]:=FALSE;
		HMI_上样轴5Z轴.execute[n]:=FALSE;
		HMI_上样轴5Z轴.write[n]:=FALSE;	
	END_FOR
		HMI_HandWheel_3Y:=FALSE;
		HMI_HandWheel_4X:=FALSE;
		HMI_HandWheel_5Z:=FALSE;
		HMI_HandWheel_6X:=FALSE;
		HMI_HandWheel_7Y:=FALSE;
		HMI_HandWheel_8Y:=FALSE;
		HMI_HandWheel_9X:=FALSE;
		HMI_HandWheel_10Z:=FALSE;
		HMI_HandWheel_11Y:=FALSE;

	
END_IF

ACTION 伺服一键回原点:
//回零请求边沿: 手动按钮=全11轴 / 开机自动=仅上样组4X5Z; 边沿触发避免每扫描复位状态机
R_TRIG_HomeAll(CLK := 一键回原点 AND MODE_State<>1 AND NOT ManualAuto);
R_TRIG_Home45(CLK := bAutoHomeReq AND MODE_State<>1);

IF R_TRIG_HomeAll.Q THEN     // 手动一键回原点: 初始化全部(并行轴 + 刮板组 + 上样组含3Y)
	玻璃上料轴1ZDATE.xHome := TRUE;
	玻璃上料轴2ZDATE.xHome := TRUE;
	刮板轴10ZDATE.xHome := TRUE;
	点样轴6XDATE.xHome := TRUE;
	点样轴7YDATE.xHome := TRUE;
	地轨轴11YDATE.xHome := TRUE;
	HOME_1STEP := 1;
	HOME_2STEP := 1;
	bAutoHomeOnly45 := FALSE;
END_IF
IF R_TRIG_Home45.Q THEN      // 开机自动: 仅初始化上样组(5Z->4X), 跳过3Y与其他轴
	HOME_2STEP := 1;
	bAutoHomeOnly45 := TRUE;
END_IF

IF 一键回原点 OR bAutoHomeReq THEN   // 仅在请求有效期运行状态机
	IF 玻璃上料轴1ZDATE.bHomed THEN 玻璃上料轴1ZDATE.xHome := FALSE; END_IF
	IF 玻璃上料轴2ZDATE.bHomed THEN 玻璃上料轴2ZDATE.xHome := FALSE; END_IF
	IF 点样轴6XDATE.bHomed THEN 点样轴6XDATE.xHome := FALSE; END_IF
	IF 点样轴7YDATE.bHomed THEN 点样轴7YDATE.xHome := FALSE; END_IF
	IF 地轨轴11YDATE.bHomed THEN 地轨轴11YDATE.xHome := FALSE; END_IF

	//刮板拍照回原点流程(仅手动): 10Z 回零后 9X,8Y
	CASE HOME_1STEP OF
		1 :
			IF 刮板轴10ZDATE.bHomed THEN
				刮板轴10ZDATE.xHome := FALSE;
				刮板轴9XDATE.xHome := TRUE;
				拍照轴8YDATE.xHome := TRUE;
				HOME_1STEP := 2;
			END_IF
		2 :
			IF 刮板轴9XDATE.bHomed THEN 刮板轴9XDATE.xHome := FALSE; END_IF
			IF 拍照轴8YDATE.bHomed THEN 拍照轴8YDATE.xHome := FALSE; END_IF
			IF 刮板轴10ZDATE.bHomed AND 刮板轴9XDATE.bHomed THEN HOME_1STEP := 0; END_IF
	END_CASE

	//上样点样回原点流程: 先 5Z(退避->回零), 再 4X(退避->回零); 严格 5Z 回零且安全高度后 4X 才动(防撞针)
	//3Y 仅手动模式(NOT bAutoHomeOnly45)在 5Z 后回零
	CASE HOME_2STEP OF
		1 :
			上样轴5Z轴DATE.xHome := FALSE;
			上样轴4X轴DATE.xHome := FALSE;
			上样轴5Z轴DATE.xMoveRel := FALSE;
			上样轴4X轴DATE.xMoveRel := FALSE;
			HOME_2STEP := 2;
		2 :
			上样轴5Z轴DATE.fRelTarget := 10.0;
			上样轴5Z轴DATE.fVelocity := 5.0;
			上样轴5Z轴DATE.xMoveRel := TRUE;
			HOME_2STEP := 3;
		3 :
			IF 上样轴5Z轴DATE.bReMoveDone THEN
				上样轴5Z轴DATE.xMoveRel := FALSE;
				上样轴5Z轴DATE.xHome := TRUE;
				HOME_2STEP := 4;
			END_IF
		4 :
			IF 上样轴5Z轴DATE.bHomed THEN
				上样轴5Z轴DATE.xHome := FALSE;
				IF NOT bAutoHomeOnly45 THEN
					打样瓶上料轴3YDATE.xHome := TRUE;
				END_IF
				IF 上样轴5Z轴DATE.fActPos < 3 THEN
					上样轴4X轴DATE.fRelTarget := 10.0;
					上样轴4X轴DATE.fVelocity := 5.0;
					上样轴4X轴DATE.xMoveRel := TRUE;
					HOME_2STEP := 5;
				END_IF
			END_IF
		5 :
			IF 上样轴4X轴DATE.bReMoveDone THEN
				上样轴4X轴DATE.xMoveRel := FALSE;
				上样轴4X轴DATE.xHome := TRUE;
				HOME_2STEP := 6;
			END_IF
		6 :
			IF 上样轴4X轴DATE.bHomed THEN 上样轴4X轴DATE.xHome := FALSE; END_IF
			IF NOT bAutoHomeOnly45 THEN
				IF 打样瓶上料轴3YDATE.bHomed THEN 打样瓶上料轴3YDATE.xHome := FALSE; END_IF
			END_IF
			IF (bAutoHomeOnly45 OR 打样瓶上料轴3YDATE.bHomed) AND 上样轴4X轴DATE.bHomed THEN
				HOME_2STEP := 0;
			END_IF
	END_CASE
END_IF

//手动一键回原点完成(全11轴回零)清请求
IF 玻璃上料轴1ZDATE.bHomed AND 玻璃上料轴2ZDATE.bHomed AND 点样轴6XDATE.bHomed AND 点样轴7YDATE.bHomed AND 地轨轴11YDATE.bHomed AND 刮板轴10ZDATE.bHomed AND 刮板轴9XDATE.bHomed AND 上样轴5Z轴DATE.bHomed AND 上样轴4X轴DATE.bHomed AND 拍照轴8YDATE.bHomed AND 打样瓶上料轴3YDATE.bHomed THEN
	一键回原点 := FALSE;
END_IF
END_ACTION

ACTION 伺服调用:
//玻璃上料轴1Z伺服控制
FB_SERVOAXIS_0(
	AXIS:= 玻璃上料轴1Z ,                    //轴名称
	xEnable:=急停  ,                         //轴使能
	xHome:= 玻璃上料轴1ZDATE.xHome,          //轴回零命令
	xJogPos:=玻璃上料轴1ZDATE.xJogPos OR Z1JOG_pos  ,     //轴正转命令
	xJogNeg:=玻璃上料轴1ZDATE.xJogNeg OR Z1JOG_neg ,     //轴反转命令
	xStop:= 玻璃上料轴1ZDATE.xStop ,         //轴停止命令
	xMoveAbs:= 玻璃上料轴1ZDATE.xMoveAbs ,   //轴绝对定位命令
	xMoveRel:= 玻璃上料轴1ZDATE.xMoveRel,    //轴相对定位命令
	XReset:= 玻璃上料轴1ZDATE.XReset OR 复位 OR bSysReset ,       //轴复位
	fAbsTarget:= 玻璃上料轴1ZDATE.fAbsTarget ,  //轴绝对定位距离
	fRelTarget:=玻璃上料轴1ZDATE.fRelTarget  ,  //轴相对移动距离
	fVelocity:= 玻璃上料轴1ZDATE.fVelocity ,    //轴定位速度
	fAcc:=1000.0 ,              //轴加速度
	fDec:= 1000.0,              //轴减速度
	fJogVel:= 15.0 ,        //轴JOG速度
	bEnabled=> 玻璃上料轴1ZDATE.bEnabled ,      //轴使能完成
	bHomed=> 回零完成1Z ,          //轴回原点完成
	bBusy=> 玻璃上料轴1ZDATE.bBusy ,            //轴运行中
	bError=> 玻璃上料轴1ZDATE.bError ,          //轴错误
	iErrorCode=>玻璃上料轴1ZDATE.iErrorCode  ,  //轴错误代码
	fActPos=>玻璃上料轴1ZDATE.fActPos  ,        //轴当前位置
	fActVel=>玻璃上料轴1ZDATE.fActVel  ,        //轴当前速度
	bAbMoveDone=>玻璃上料轴1ZDATE.bAbMoveDone ,  //轴绝对定位完成
	bReMoveDone =>玻璃上料轴1ZDATE.bReMoveDone ,);    //轴相对定位完成 
玻璃上料轴1ZDATE.bHomed S= 回零完成1Z;
IF  玻璃上料轴1ZDATE.xHome THEN
	玻璃上料轴1ZDATE.bHomed:=FALSE;
END_IF

//玻璃上料轴2Z伺服控制
FB_SERVOAXIS_1(
	AXIS:= 玻璃上料轴2Z ,                    //轴名称
	xEnable:=急停  ,                         //轴使能
	xHome:= 玻璃上料轴2ZDATE.xHome,          //轴回零命令
	xJogPos:=玻璃上料轴2ZDATE.xJogPos OR Z2JOG_POS ,     //轴正转命令
	xJogNeg:=玻璃上料轴2ZDATE.xJogNeg OR Z2JOG_NEG ,     //轴反转命令
	xStop:= 玻璃上料轴2ZDATE.xStop ,         //轴停止命令
	xMoveAbs:= 玻璃上料轴2ZDATE.xMoveAbs ,   //轴绝对定位命令
	xMoveRel:= 玻璃上料轴2ZDATE.xMoveRel,    //轴相对定位命令
	XReset:= 玻璃上料轴2ZDATE.XReset OR 复位 OR bSysReset ,       //轴复位
	fAbsTarget:= 玻璃上料轴2ZDATE.fAbsTarget ,  //轴绝对定位距离
	fRelTarget:=玻璃上料轴2ZDATE.fRelTarget  ,  //轴相对移动距离
	fVelocity:= 玻璃上料轴2ZDATE.fVelocity ,    //轴定位速度
	fAcc:=1000.0 ,              //轴加速度
	fDec:= 1000.0,              //轴减速度
	fJogVel:= 15.0 ,        //轴JOG速度
	bEnabled=> 玻璃上料轴2ZDATE.bEnabled ,      //轴使能完成
	bHomed=> 回零完成2Z ,          //轴回原点完成
	bBusy=> 玻璃上料轴2ZDATE.bBusy ,            //轴运行中
	bError=> 玻璃上料轴2ZDATE.bError ,          //轴错误
	iErrorCode=>玻璃上料轴2ZDATE.iErrorCode  ,  //轴错误代码
	fActPos=>玻璃上料轴2ZDATE.fActPos  ,        //轴当前位置
	fActVel=>玻璃上料轴2ZDATE.fActVel  ,        //轴当前速度
	bAbMoveDone=>玻璃上料轴2ZDATE.bAbMoveDone ,  //轴绝对定位完成
	bReMoveDone =>玻璃上料轴2ZDATE.bReMoveDone ,);    //轴相对定位完成 
玻璃上料轴2ZDATE.bHomed S= 回零完成2Z;
IF  玻璃上料轴2ZDATE.xHome THEN
	玻璃上料轴2ZDATE.bHomed:=FALSE;
END_IF	
	
FB_SERVOAXIS_2(
	AXIS:= 打样瓶上料轴3Y ,                    //轴名称
	xEnable:= 急停 AND NOT (Sampling_Servo_FreeMove AND (上样轴5Z轴DATE.fActPos < 3)) ,   //轴使能(去使能手推: 仅5Z抬起<3时放开3Y)
	xHome:= 打样瓶上料轴3YDATE.xHome,          //轴回零命令
	xJogPos:=打样瓶上料轴3YDATE.xJogPos  ,     //轴正转命令
	xJogNeg:=打样瓶上料轴3YDATE.xJogNeg  ,     //轴反转命令
	xStop:= 打样瓶上料轴3YDATE.xStop ,         //轴停止命令
	xMoveAbs:= 打样瓶上料轴3YDATE.xMoveAbs ,   //轴绝对定位命令
	xMoveRel:= 打样瓶上料轴3YDATE.xMoveRel,    //轴相对定位命令
	XReset:= 打样瓶上料轴3YDATE.XReset OR 复位 OR bSysReset,       //轴复位
	fAbsTarget:= 打样瓶上料轴3YDATE.fAbsTarget ,  //轴绝对定位距离
	fRelTarget:=打样瓶上料轴3YDATE.fRelTarget  ,  //轴相对移动距离
	fVelocity:= 打样瓶上料轴3YDATE.fVelocity ,    //轴定位速度
	fAcc:=500.0 ,              //轴加速度
	fDec:= 500.0 ,              //轴减速度
	fJogVel:= 50.0 ,        //轴JOG速度
	bEnabled=> 打样瓶上料轴3YDATE.bEnabled ,      //轴使能完成
	bHomed=> 回零完成3Y ,          //轴回原点完成
	bBusy=> 打样瓶上料轴3YDATE.bBusy ,            //轴运行中
	bError=> 打样瓶上料轴3YDATE.bError ,          //轴错误
	iErrorCode=>打样瓶上料轴3YDATE.iErrorCode  ,  //轴错误代码
	fActPos=>打样瓶上料轴3YDATE.fActPos  ,        //轴当前位置
	fActVel=>打样瓶上料轴3YDATE.fActVel  ,        //轴当前速度
	bAbMoveDone=>打样瓶上料轴3YDATE.bAbMoveDone ,  //轴绝对定位完成
	bReMoveDone =>打样瓶上料轴3YDATE.bReMoveDone ,);    //轴相对定位完成 
打样瓶上料轴3YDATE.bHomed S= 回零完成3Y;
IF  打样瓶上料轴3YDATE.xHome THEN
	打样瓶上料轴3YDATE.bHomed:=FALSE;
END_IF		

//点样轴6X伺服控制
FB_SERVOAXIS_3(
	AXIS:= 点样轴6X ,                    //轴名称
	xEnable:=急停  ,                         //轴使能
	xHome:= 点样轴6XDATE.xHome,          //轴回零命令
	xJogPos:=点样轴6XDATE.xJogPos  ,     //轴正转命令
	xJogNeg:=点样轴6XDATE.xJogNeg  ,     //轴反转命令
	xStop:= 点样轴6XDATE.xStop ,         //轴停止命令
	xMoveAbs:= 点样轴6XDATE.xMoveAbs ,   //轴绝对定位命令
	xMoveRel:= 点样轴6XDATE.xMoveRel,    //轴相对定位命令
	XReset:= 点样轴6XDATE.XReset OR 复位 OR bSysReset,       //轴复位
	fAbsTarget:= 点样轴6XDATE.fAbsTarget ,  //轴绝对定位距离
	fRelTarget:=点样轴6XDATE.fRelTarget  ,  //轴相对移动距离
	fVelocity:= 点样轴6XDATE.fVelocity ,    //轴定位速度
	fAcc:=5500.0 ,              //轴加速度
	fDec:= 5500.0,              //轴减速度
	fJogVel:= 50.0 ,        //轴JOG速度
	bEnabled=> 点样轴6XDATE.bEnabled ,      //轴使能完成
	bHomed=> 回零完成6X ,          //轴回原点完成
	bBusy=> 点样轴6XDATE.bBusy ,            //轴运行中
	bError=> 点样轴6XDATE.bError ,          //轴错误
	iErrorCode=>点样轴6XDATE.iErrorCode  ,  //轴错误代码
	fActPos=>点样轴6XDATE.fActPos  ,        //轴当前位置
	fActVel=>点样轴6XDATE.fActVel  ,        //轴当前速度
	bAbMoveDone=>点样轴6XDATE.bAbMoveDone ,  //轴绝对定位完成
	bReMoveDone =>点样轴6XDATE.bReMoveDone ,);    //轴相对定位完成 
点样轴6XDATE.bHomed S=回零完成6X;
IF  点样轴6XDATE.xHome THEN
	点样轴6XDATE.bHomed:=FALSE;
END_IF

//点样轴7Y伺服控制
FB_SERVOAXIS_4(
	AXIS:= 点样轴7Y ,                    //轴名称
	xEnable:=急停  ,                         //轴使能
	xHome:= 点样轴7YDATE.xHome,          //轴回零命令
	xJogPos:=点样轴7YDATE.xJogPos  ,     //轴正转命令
	xJogNeg:=点样轴7YDATE.xJogNeg  ,     //轴反转命令
	xStop:= 点样轴7YDATE.xStop ,         //轴停止命令
	xMoveAbs:= 点样轴7YDATE.xMoveAbs ,   //轴绝对定位命令
	xMoveRel:= 点样轴7YDATE.xMoveRel,    //轴相对定位命令
	XReset:= 点样轴7YDATE.XReset OR 复位 OR bSysReset,       //轴复位
	fAbsTarget:= 点样轴7YDATE.fAbsTarget ,  //轴绝对定位距离
	fRelTarget:=点样轴7YDATE.fRelTarget  ,  //轴相对移动距离
	fVelocity:= 点样轴7YDATE.fVelocity ,    //轴定位速度
	fAcc:=500.0 ,              //轴加速度
	fDec:= 500.0 ,              //轴减速度
	fJogVel:= 50.0 ,        //轴JOG速度
	bEnabled=> 点样轴7YDATE.bEnabled ,      //轴使能完成
	bHomed=>  回零完成7Y,          //轴回原点完成
	bBusy=> 点样轴7YDATE.bBusy ,            //轴运行中
	bError=> 点样轴7YDATE.bError ,          //轴错误
	iErrorCode=>点样轴7YDATE.iErrorCode  ,  //轴错误代码
	fActPos=>点样轴7YDATE.fActPos  ,        //轴当前位置
	fActVel=>点样轴7YDATE.fActVel  ,        //轴当前速度
	bAbMoveDone=>点样轴7YDATE.bAbMoveDone ,  //轴绝对定位完成
	bReMoveDone =>点样轴7YDATE.bReMoveDone ,);    //轴相对定位完成 
点样轴7YDATE.bHomed S=回零完成7Y;
IF  点样轴7YDATE.xHome THEN
	点样轴7YDATE.bHomed:=FALSE;
END_IF

//拍照轴8Y伺服控制
FB_SERVOAXIS_5(
	AXIS:= 拍照轴8Y ,                    //轴名称
	xEnable:=急停  ,                         //轴使能
	xHome:= 拍照轴8YDATE.xHome,          //轴回零命令
	xJogPos:=拍照轴8YDATE.xJogPos  ,     //轴正转命令
	xJogNeg:=拍照轴8YDATE.xJogNeg  ,     //轴反转命令
	xStop:= 拍照轴8YDATE.xStop ,         //轴停止命令
	xMoveAbs:= 拍照轴8YDATE.xMoveAbs AND  刮板拍照遮光气缸上位 AND 刮板轴10ZDATE.fActPos<6 ,   //轴绝对定位命令
	xMoveRel:= 拍照轴8YDATE.xMoveRel,    //轴相对定位命令
	XReset:= 拍照轴8YDATE.XReset OR 复位 OR bSysReset,       //轴复位
	fAbsTarget:= 拍照轴8YDATE.fAbsTarget ,  //轴绝对定位距离
	fRelTarget:=拍照轴8YDATE.fRelTarget  ,  //轴相对移动距离
	fVelocity:= 拍照轴8YDATE.fVelocity ,    //轴定位速度
	fAcc:=500.0 ,              //轴加速度
	fDec:= 500.0 ,              //轴减速度
	fJogVel:= 50.0 ,        //轴JOG速度
	bEnabled=> 拍照轴8YDATE.bEnabled ,      //轴使能完成
	bHomed=> 回零完成8Y ,          //轴回原点完成
	bBusy=> 拍照轴8YDATE.bBusy ,            //轴运行中
	bError=> 拍照轴8YDATE.bError ,          //轴错误
	iErrorCode=>拍照轴8YDATE.iErrorCode  ,  //轴错误代码
	fActPos=>拍照轴8YDATE.fActPos  ,        //轴当前位置
	fActVel=>拍照轴8YDATE.fActVel  ,        //轴当前速度
	bAbMoveDone=>拍照轴8YDATE.bAbMoveDone ,  //轴绝对定位完成
	bReMoveDone =>拍照轴8YDATE.bReMoveDone ,);    //轴相对定位完成 
	拍照轴8YDATE.bHomed S=回零完成8Y;
IF  拍照轴8YDATE.xHome THEN
	拍照轴8YDATE.bHomed:=FALSE;
END_IF

//刮板轴9X伺服控制
FB_SERVOAXIS_6(
	AXIS:= 刮板轴9X ,                    //轴名称
	xEnable:=急停  ,                         //轴使能
	xHome:= 刮板轴9XDATE.xHome,          //轴回零命令
	xJogPos:=刮板轴9XDATE.xJogPos  ,     //轴正转命令
	xJogNeg:=刮板轴9XDATE.xJogNeg  ,     //轴反转命令
	xStop:= 刮板轴9XDATE.xStop ,         //轴停止命令
	xMoveAbs:= 刮板轴9XDATE.xMoveAbs AND  刮板轴10ZDATE.fActPos<6,   //轴绝对定位命令
	xMoveRel:= 刮板轴9XDATE.xMoveRel,    //轴相对定位命令
	XReset:= 刮板轴9XDATE.XReset OR 复位 OR bSysReset,       //轴复位
	fAbsTarget:= 刮板轴9XDATE.fAbsTarget  ,  //轴绝对定位距离
	fRelTarget:=刮板轴9XDATE.fRelTarget  ,  //轴相对移动距离
	fVelocity:= 刮板轴9XDATE.fVelocity ,    //轴定位速度
	fAcc:=500.0 ,              //轴加速度
	fDec:= 500.0 ,              //轴减速度
	fJogVel:= 50.0 ,        //轴JOG速度
	bEnabled=> 刮板轴9XDATE.bEnabled ,      //轴使能完成
	bHomed=>  回零完成9X,          //轴回原点完成
	bBusy=> 刮板轴9XDATE.bBusy ,            //轴运行中
	bError=> 刮板轴9XDATE.bError ,          //轴错误
	iErrorCode=>刮板轴9XDATE.iErrorCode  ,  //轴错误代码
	fActPos=>刮板轴9XDATE.fActPos  ,        //轴当前位置
	fActVel=>刮板轴9XDATE.fActVel  ,        //轴当前速度
	bAbMoveDone=>刮板轴9XDATE.bAbMoveDone ,  //轴绝对定位完成
	bReMoveDone =>刮板轴9XDATE.bReMoveDone ,);    //轴相对定位完成 
刮板轴9XDATE.bHomed S= 回零完成9X;
IF  刮板轴9XDATE.xHome THEN
	刮板轴9XDATE.bHomed:=FALSE;
END_IF

//刮板轴10Z伺服控制
FB_SERVOAXIS_7(
	AXIS:= 刮板轴10Z ,                    //轴名称
	xEnable:=急停  ,                         //轴使能
	xHome:= 刮板轴10ZDATE.xHome,          //轴回零命令
	xJogPos:=刮板轴10ZDATE.xJogPos  ,     //轴正转命令
	xJogNeg:=刮板轴10ZDATE.xJogNeg  ,     //轴反转命令
	xStop:= 刮板轴10ZDATE.xStop ,         //轴停止命令
	xMoveAbs:= 刮板轴10ZDATE.xMoveAbs ,   //轴绝对定位命令
	xMoveRel:= 刮板轴10ZDATE.xMoveRel,    //轴相对定位命令
	XReset:= 刮板轴10ZDATE.XReset OR 复位 OR bSysReset,       //轴复位
	fAbsTarget:= 刮板轴10ZDATE.fAbsTarget ,  //轴绝对定位距离
	fRelTarget:=刮板轴10ZDATE.fRelTarget  ,  //轴相对移动距离
	fVelocity:= 刮板轴10ZDATE.fVelocity ,    //轴定位速度
	fAcc:=500.0  ,              //轴加速度
	fDec:= 500.0 ,              //轴减速度
	fJogVel:= 50.0 ,        //轴JOG速度
	bEnabled=> 刮板轴10ZDATE.bEnabled ,      //轴使能完成
	bHomed=> 回零完成10Z ,          //轴回原点完成
	bBusy=> 刮板轴10ZDATE.bBusy ,            //轴运行中
	bError=> 刮板轴10ZDATE.bError ,          //轴错误
	iErrorCode=>刮板轴10ZDATE.iErrorCode  ,  //轴错误代码
	fActPos=>刮板轴10ZDATE.fActPos  ,        //轴当前位置
	fActVel=>刮板轴10ZDATE.fActVel  ,        //轴当前速度
	bAbMoveDone=>刮板轴10ZDATE.bAbMoveDone ,  //轴绝对定位完成
	bReMoveDone =>刮板轴10ZDATE.bReMoveDone ,);    //轴相对定位完成 
刮板轴10ZDATE.bHomed S= 回零完成10Z;
IF  刮板轴10ZDATE.xHome THEN
	刮板轴10ZDATE.bHomed:=FALSE;
END_IF	
	
//地轨轴11Y伺服控制
FB_SERVOAXIS_8(
	AXIS:= 地轨轴11Y ,                    //轴名称
	xEnable:=急停  ,                         //轴使能
	xHome:= 地轨轴11YDATE.xHome,          //轴回零命令
	xJogPos:=地轨轴11YDATE.xJogPos  ,     //轴正转命令
	xJogNeg:=地轨轴11YDATE.xJogNeg  ,     //轴反转命令
	xStop:= 地轨轴11YDATE.xStop ,         //轴停止命令
	xMoveAbs:= 地轨轴11YDATE.xMoveAbs  ,   //轴绝对定位命令
	xMoveRel:= 地轨轴11YDATE.xMoveRel,    //轴相对定位命令
	XReset:= 地轨轴11YDATE.XReset OR 复位 OR bSysReset,       //轴复位
	fAbsTarget:= 地轨轴11YDATE.fAbsTarget ,  //轴绝对定位距离
	fRelTarget:=地轨轴11YDATE.fRelTarget  ,  //轴相对移动距离
	fVelocity:= 地轨轴11YDATE.fVelocity ,    //轴定位速度
	fAcc:=500.0 ,              //轴加速度
	fDec:= 500.0 ,              //轴减速度
	fJogVel:= 50.0 ,        //轴JOG速度
	bEnabled=> 地轨轴11YDATE.bEnabled ,      //轴使能完成
	bHomed=>  回零完成11Y,          //轴回原点完成
	bBusy=> 地轨轴11YDATE.bBusy ,            //轴运行中
	bError=> 地轨轴11YDATE.bError ,          //轴错误
	iErrorCode=>地轨轴11YDATE.iErrorCode  ,  //轴错误代码
	fActPos=>地轨轴11YDATE.fActPos  ,        //轴当前位置
	fActVel=>地轨轴11YDATE.fActVel  ,        //轴当前速度
	bAbMoveDone=>地轨轴11YDATE.bAbMoveDone ,  //轴绝对定位完成
	bReMoveDone =>地轨轴11YDATE.bReMoveDone ,);    //轴相对定位完成 
地轨轴11YDATE.bHomed S=回零完成11Y;
IF  地轨轴11YDATE.xHome THEN
	地轨轴11YDATE.bHomed:=FALSE;
END_IF

//上样轴4X轴伺服控制
FB_SERVOAXIS_9(
	AXIS:= 上样轴4X轴 ,                    //轴名称
	xEnable:= 急停 AND NOT (Sampling_Servo_FreeMove AND (上样轴5Z轴DATE.fActPos < 3)) ,   //轴使能(去使能手推: 仅5Z抬起<3时放开4X)
	xHome:= 上样轴4X轴DATE.xHome,          //轴回零命令
	xJogPos:=上样轴4X轴DATE.xJogPos  ,     //轴正转命令
	xJogNeg:=上样轴4X轴DATE.xJogNeg  ,     //轴反转命令
	xStop:= 上样轴4X轴DATE.xStop ,         //轴停止命令
	xMoveAbs:= 上样轴4X轴DATE.xMoveAbs AND  上样轴5Z轴DATE.fActPos<3 ,   //轴绝对定位命令
	xMoveRel:= 上样轴4X轴DATE.xMoveRel AND  上样轴5Z轴DATE.fActPos<3,    //轴相对定位命令
	XReset:= 上样轴4X轴DATE.XReset OR 复位 OR bSysReset,       //轴复位
	fAbsTarget:= 上样轴4X轴DATE.fAbsTarget ,  //轴绝对定位距离
	fRelTarget:=上样轴4X轴DATE.fRelTarget  ,  //轴相对移动距离
	fVelocity:= 上样轴4X轴DATE.fVelocity ,    //轴定位速度
	fAcc:=200.0 ,              //轴加速度
	fDec:= 200.0 ,              //轴减速度
	fJogVel:= 5.0,        //轴JOG速度
	bEnabled=> 上样轴4X轴DATE.bEnabled ,      //轴使能完成
	bHomed=>  回零完成4X,          //轴回原点完成
	bBusy=> 上样轴4X轴DATE.bBusy ,            //轴运行中
	bError=> 上样轴4X轴DATE.bError ,          //轴错误
	iErrorCode=>上样轴4X轴DATE.iErrorCode  ,  //轴错误代码
	fActPos=>上样轴4X轴DATE.fActPos  ,        //轴当前位置
	fActVel=>上样轴4X轴DATE.fActVel  ,        //轴当前速度
	bAbMoveDone=>上样轴4X轴DATE.bAbMoveDone ,  //轴绝对定位完成
	bReMoveDone =>上样轴4X轴DATE.bReMoveDone ,);    //轴相对定位完成 
上样轴4X轴DATE.bHomed S=回零完成4X;
	%QB2216:= 27;             //回零模式27
IF NOT  急停 OR 上样轴4X轴DATE.xHome THEN
	上样轴4X轴DATE.bHomed:=FALSE;
END_IF

//上样轴5Z轴伺服控制
FB_SERVOAXIS_10(
	AXIS:= 上样轴5Z轴 ,                    //轴名称
	xEnable:=急停  ,                         //轴使能
	xHome:= 上样轴5Z轴DATE.xHome,          //轴回零命令
	xJogPos:=上样轴5Z轴DATE.xJogPos  ,     //轴正转命令
	xJogNeg:=上样轴5Z轴DATE.xJogNeg  ,     //轴反转命令
	xStop:= 上样轴5Z轴DATE.xStop ,         //轴停止命令
	xMoveAbs:= 上样轴5Z轴DATE.xMoveAbs ,   //轴绝对定位命令
	xMoveRel:= 上样轴5Z轴DATE.xMoveRel,    //轴相对定位命令
	XReset:= 上样轴5Z轴DATE.XReset OR 复位 OR bSysReset ,       //轴复位
	fAbsTarget:= 上样轴5Z轴DATE.fAbsTarget ,  //轴绝对定位距离
	fRelTarget:=上样轴5Z轴DATE.fRelTarget  ,  //轴相对移动距离
	fVelocity:= 上样轴5Z轴DATE.fVelocity ,    //轴定位速度
	fAcc:=300.0  ,              //轴加速度
	fDec:= 300.0 ,              //轴减速度
	fJogVel:= 20.0 ,        //轴JOG速度
	bEnabled=> 上样轴5Z轴DATE.bEnabled ,      //轴使能完成
	bHomed=> 回零完成5Z ,          //轴回原点完成
	bBusy=> 上样轴5Z轴DATE.bBusy ,            //轴运行中
	bError=> 上样轴5Z轴DATE.bError ,          //轴错误
	iErrorCode=>上样轴5Z轴DATE.iErrorCode  ,  //轴错误代码
	fActPos=>上样轴5Z轴DATE.fActPos  ,        //轴当前位置
	fActVel=>上样轴5Z轴DATE.fActVel  ,        //轴当前速度
	bAbMoveDone=>上样轴5Z轴DATE.bAbMoveDone ,   //轴绝对定位完成
	bReMoveDone =>上样轴5Z轴DATE.bReMoveDone , );   //轴相对定位完成 
上样轴5Z轴DATE.bHomed S=回零完成5Z;
	%QB2228:= 27;                 //回零模式27
IF NOT  急停 OR 上样轴5Z轴DATE.xHome THEN
	上样轴5Z轴DATE.bHomed:=FALSE;
END_IF

//上样4X 与 打样3Y 实际使能镜像 -> 供上位机标定页显示真状态 (去使能手推时为 FALSE)
Sampling_Servo_Enabled := 上样轴4X轴DATE.bEnabled AND 打样瓶上料轴3YDATE.bEnabled;
END_ACTION

ACTION 位置示教:

//打样瓶上料轴3Y位置示教
FB_Teach_1(HMI_Servo:=HMI_打样瓶上料轴3Y , 
			Servo:=打样瓶上料轴3YDATE );
//点样轴6X位置示教
FB_Teach_2(HMI_Servo:=HMI_点样轴6X , 
			Servo:=点样轴6XDATE );
//点样轴7Y位置示教
FB_Teach_3(HMI_Servo:=HMI_点样轴7Y , 
			Servo:=点样轴7YDATE );			
//地轨轴11Y位置示教
FB_Teach_4(HMI_Servo:=HMI_地轨轴11Y , 
			Servo:=地轨轴11YDATE );			
//上样轴4X轴位置示教
FB_Teach_5(HMI_Servo:=HMI_上样轴4X轴 , 
			Servo:=上样轴4X轴DATE );			
//上样轴5Z轴位置示教
FB_Teach_6(HMI_Servo:=HMI_上样轴5Z轴 , 
			Servo:=上样轴5Z轴DATE );
END_ACTION

END_PROGRAM

// Device/Application/25_FB_功能块/FB_SERVOAXIS
FUNCTION_BLOCK FB_SERVOAXIS
VAR_IN_OUT
	AXIS: AXIS_REF_SM3;
END_VAR
VAR_INPUT
    // 轴控制命令
	// 轴使能
    xEnable    : BOOL;  // 轴使能
    xHome      : BOOL;  // 回原点命令
    xJogPos    : BOOL;  // 正方向点动
    xJogNeg    : BOOL;  // 负方向点动
    xStop      : BOOL;  // 停止命令
    xMoveAbs   : BOOL;  // 绝对运动启动
    xMoveRel   : BOOL;  // 相对运动启动
	XReset:BOOL; //轴复位
    
    // 运动参数
    fAbsTarget  : LREAL := 0.0;  // 绝对位置目标
    fRelTarget  : LREAL := 0.0;  // 相对运动距离
    fVelocity   : LREAL := 100.0;  // 运行速度
    fAcc        : LREAL := 1000.0;  // 加速度
    fDec        : LREAL := 1000.0;  // 减速度
    fJogVel     : LREAL := 50.0;  // 点动速度 
END_VAR
VAR_OUTPUT
    bEnabled    : BOOL;  // 轴使能状态
    bHomed      : BOOL;  // 原点完成
    bBusy       : BOOL;  // 轴忙状态
    bError      : BOOL;  // 轴报警
    iErrorCode  : DINT;  // 错误代码
    fActPos     : LREAL;  // 实际位置
    fActVel     : LREAL;  // 实际速度
    bAbMoveDone   : BOOL;  // 运动完成
	// 轴使能
	bReMoveDone: BOOL;
END_VAR
VAR
    // 运动控制实例
     MC_Power   : MC_Power;    // 轴使能
     MC_Home    : MC_Home;     // 回原点
	// 停止
	MC_Homing: MC_Home;
     MC_Halt    : MC_Halt;     // 停止
     MC_MoveAbsolute : MC_MoveAbsolute;  // 绝对定位
     MC_MoveRelative : MC_MoveRelative;  // 相对定位
     MC_Jog : MC_Jog ;  // 点动
	 MC_Reset:MC_Reset; //轴复位
    
    // 内部变量
    bAxisEnabled : BOOL := FALSE;  // 轴使能标志
    bHomeDone    : BOOL := FALSE;  // 回零完成标志
    bMoving      : BOOL := FALSE;  // 运动中标志
    bHoming      : BOOL := FALSE;  // 回零中标志 
END_VAR

//轴使能
MC_Power(
	Axis:=AXIS   , 
	Enable:= TRUE  , 
	bRegulatorOn:= xEnable , 
	bDriveStart:=TRUE  , 
	Status=> bEnabled  , 
	bRegulatorRealState=> , 
	bDriveStartRealState=> , 
	Busy=> , 
	Error=>  , 
	ErrorID=>  );
//轴回零
MC_Home(
	Axis:= AXIS, 
	Execute:= xHome , 
	Position:= , 
	Done=> bHomed , 
	Busy=> bHoming , 
	CommandAborted=> , 
	Error=> , 
	ErrorID=> );

